LIN {X 0.053,Y -418.660,Z 515.534,A 0.000,B 0.000,C 90.000,E1 132.123} C_DIS
LIN {X -0.078,Y -417.973,Z 515.527,A 0.000,B 0.000,C 90.000,E1 130.782} C_DIS
LIN {X -0.019,Y -416.880,Z 515.517,A 0.000,B 0.000,C 90.000,E1 129.072} C_DIS
LIN {X -0.176,Y -415.818,Z 515.510,A 0.000,B 0.000,C 90.000,E1 127.729} C_DIS
LIN {X 0.148,Y -414.723,Z 515.501,A 0.000,B 0.000,C 90.000,E1 126.217} C_DIS
LIN {X 0.110,Y -414.727,Z 515.501,A 0.000,B 0.000,C 90.000,E1 126.217} C_DIS
LIN {X -0.098,Y -415.454,Z 515.500,A 0.000,B 0.000,C 90.000,E1 126.011} C_DIS
LIN {X -0.035,Y -425.850,Z 515.477,A 0.000,B 0.000,C 90.000,E1 121.926} C_DIS
LIN {X -0.091,Y -430.874,Z 515.468,A 0.000,B 0.000,C 90.000,E1 120.256} C_DIS
LIN {X -0.162,Y -439.919,Z 515.448,A 0.000,B 0.000,C 90.000,E1 116.616} C_DIS
LIN {X 0.024,Y -444.712,Z 515.439,A 0.000,B 0.000,C 90.000,E1 114.951} C_DIS
LIN {X -0.004,Y -454.683,Z 515.415,A 0.000,B 0.000,C 90.000,E1 110.737} C_DIS
LIN {X -0.228,Y -456.616,Z 515.411,A 0.000,B 0.000,C 90.000,E1 110.066} C_DIS
LIN {X -0.262,Y -456.708,Z 515.411,A 0.000,B 0.000,C 90.000,E1 110.066} C_DIS
LIN {X 0.078,Y -489.584,Z 515.405,A 0.000,B 0.000,C 90.000,E1 108.960} C_DIS
LIN {X 0.012,Y -503.421,Z 515.403,A 0.000,B 0.000,C 90.000,E1 108.489} C_DIS
LIN {X -0.146,Y -520.802,Z 515.399,A 0.000,B 0.000,C 90.000,E1 107.873} C_DIS
LIN {X -0.071,Y -534.501,Z 515.396,A 0.000,B 0.000,C 90.000,E1 107.330} C_DIS
LIN {X 0.020,Y -541.040,Z 515.395,A 0.000,B 0.000,C 90.000,E1 107.040} C_DIS
LIN {X 0.041,Y -547.560,Z 515.393,A 0.000,B 0.000,C 90.000,E1 106.732} C_DIS
LIN {X 0.199,Y -553.930,Z 515.391,A 0.000,B 0.000,C 90.000,E1 106.386} C_DIS
LIN {X -0.017,Y -559.838,Z 515.389,A 0.000,B 0.000,C 90.000,E1 106.079} C_DIS
LIN {X -0.116,Y -565.718,Z 515.387,A 0.000,B 0.000,C 90.000,E1 105.717} C_DIS
LIN {X -0.140,Y -571.713,Z 515.385,A 0.000,B 0.000,C 90.000,E1 105.300} C_DIS
LIN {X 0.274,Y -577.362,Z 515.383,A 0.000,B 0.000,C 90.000,E1 104.828} C_DIS
LIN {X -0.225,Y -582.899,Z 515.380,A 0.000,B 0.000,C 90.000,E1 104.411} C_DIS
LIN {X -0.192,Y -588.073,Z 515.377,A 0.000,B 0.000,C 90.000,E1 103.939} C_DIS
LIN {X 0.183,Y -593.940,Z 515.374,A 0.000,B 0.000,C 90.000,E1 103.300} C_DIS
LIN {X -0.050,Y -601.039,Z 515.370,A 0.000,B 0.000,C 90.000,E1 102.535} C_DIS
LIN {X 0.069,Y -605.510,Z 515.367,A 0.000,B 0.000,C 90.000,E1 102.007} C_DIS
LIN {X 0.219,Y -609.763,Z 515.364,A 0.000,B 0.000,C 90.000,E1 101.478} C_DIS
LIN {X 0.057,Y -615.614,Z 515.360,A 0.000,B 0.000,C 90.000,E1 100.715} C_DIS
LIN {X -0.165,Y -620.986,Z 515.355,A 0.000,B 0.000,C 90.000,E1 99.962} C_DIS
LIN {X 0.315,Y -624.961,Z 515.352,A 0.000,B 0.000,C 90.000,E1 99.321} C_DIS
LIN {X 0.189,Y -629.618,Z 515.348,A 0.000,B 0.000,C 90.000,E1 98.568} C_DIS
LIN {X 0.109,Y -633.925,Z 515.344,A 0.000,B 0.000,C 90.000,E1 97.814} C_DIS
LIN {X -0.201,Y -639.249,Z 515.338,A 0.000,B 0.000,C 90.000,E1 96.834} C_DIS
LIN {X -0.264,Y -642.915,Z 515.334,A 0.000,B 0.000,C 90.000,E1 96.087} C_DIS
LIN {X -0.054,Y -648.552,Z 515.327,A 0.000,B 0.000,C 90.000,E1 94.821} C_DIS
LIN {X -0.191,Y -652.488,Z 515.321,A 0.000,B 0.000,C 90.000,E1 93.841} C_DIS
LIN {X 0.041,Y -654.246,Z 515.319,A 0.000,B 0.000,C 90.000,E1 93.326} C_DIS
LIN {X 0.125,Y -656.498,Z 515.314,A 0.000,B 0.000,C 90.000,E1 92.579} C_DIS
LIN {X -0.263,Y -657.795,Z 515.312,A 0.000,B 0.000,C 90.000,E1 92.121} C_DIS
LIN {X 0.036,Y -658.865,Z 515.309,A 0.000,B 0.000,C 90.000,E1 91.604} C_DIS
LIN {X 0.139,Y -660.082,Z 515.305,A 0.000,B 0.000,C 90.000,E1 90.859} C_DIS
LIN {X -0.224,Y -660.593,Z 515.302,A 0.000,B 0.000,C 90.000,E1 90.401} C_DIS
LIN {X 0.256,Y -660.820,Z 515.301,A 0.000,B 0.000,C 90.000,E1 90.115} C_DIS
LIN {X -0.279,Y -660.960,Z 515.297,A 0.000,B 0.000,C 90.000,E1 89.427} C_DIS
LIN {X -0.154,Y -660.743,Z 515.293,A 0.000,B 0.000,C 90.000,E1 88.682} C_DIS
LIN {X -0.334,Y -660.657,Z 515.291,A 0.000,B 0.000,C 90.000,E1 88.453} C_DIS
LIN {X -0.193,Y -659.821,Z 515.287,A 0.000,B 0.000,C 90.000,E1 87.707} C_DIS
LIN {X 0.100,Y -659.109,Z 515.284,A 0.000,B 0.000,C 90.000,E1 87.192} C_DIS
LIN {X 0.231,Y -657.662,Z 515.280,A 0.000,B 0.000,C 90.000,E1 86.445} C_DIS
LIN {X 0.039,Y -657.169,Z 515.279,A 0.000,B 0.000,C 90.000,E1 86.216} C_DIS
LIN {X 0.152,Y -655.263,Z 515.275,A 0.000,B 0.000,C 90.000,E1 85.469} C_DIS
LIN {X -0.199,Y -653.811,Z 515.272,A 0.000,B 0.000,C 90.000,E1 85.008} C_DIS
LIN {X 0.095,Y -652.092,Z 515.269,A 0.000,B 0.000,C 90.000,E1 84.489} C_DIS
LIN {X -0.068,Y -648.360,Z 515.264,A 0.000,B 0.000,C 90.000,E1 83.514} C_DIS
LIN {X 0.026,Y -645.162,Z 515.260,A 0.000,B 0.000,C 90.000,E1 82.761} C_DIS
LIN {X 0.094,Y -641.550,Z 515.256,A 0.000,B 0.000,C 90.000,E1 82.008} C_DIS
LIN {X 0.124,Y -637.675,Z 515.252,A 0.000,B 0.000,C 90.000,E1 81.254} C_DIS
LIN {X 0.309,Y -634.940,Z 515.249,A 0.000,B 0.000,C 90.000,E1 80.735} C_DIS
LIN {X -0.208,Y -631.219,Z 515.245,A 0.000,B 0.000,C 90.000,E1 80.151} C_DIS
LIN {X -0.128,Y -627.261,Z 515.242,A 0.000,B 0.000,C 90.000,E1 79.511} C_DIS
LIN {X -0.083,Y -623.088,Z 515.238,A 0.000,B 0.000,C 90.000,E1 78.870} C_DIS
LIN {X -0.237,Y -616.739,Z 515.233,A 0.000,B 0.000,C 90.000,E1 77.993} C_DIS
LIN {X -0.288,Y -611.718,Z 515.230,A 0.000,B 0.000,C 90.000,E1 77.353} C_DIS
LIN {X -0.244,Y -606.038,Z 515.226,A 0.000,B 0.000,C 90.000,E1 76.700} C_DIS
LIN {X -0.133,Y -601.097,Z 515.223,A 0.000,B 0.000,C 90.000,E1 76.172} C_DIS
LIN {X 0.043,Y -595.900,Z 515.220,A 0.000,B 0.000,C 90.000,E1 75.644} C_DIS
LIN {X -0.173,Y -590.464,Z 515.218,A 0.000,B 0.000,C 90.000,E1 75.172} C_DIS
LIN {X -0.106,Y -584.679,Z 515.215,A 0.000,B 0.000,C 90.000,E1 74.685} C_DIS
LIN {X 0.133,Y -578.609,Z 515.212,A 0.000,B 0.000,C 90.000,E1 74.212} C_DIS
LIN {X 0.247,Y -572.611,Z 515.210,A 0.000,B 0.000,C 90.000,E1 73.795} C_DIS
LIN {X 0.100,Y -567.660,Z 515.208,A 0.000,B 0.000,C 90.000,E1 73.504} C_DIS
LIN {X -0.166,Y -562.686,Z 515.207,A 0.000,B 0.000,C 90.000,E1 73.251} C_DIS
LIN {X -0.083,Y -555.857,Z 515.205,A 0.000,B 0.000,C 90.000,E1 72.906} C_DIS
LIN {X 0.024,Y -548.840,Z 515.203,A 0.000,B 0.000,C 90.000,E1 72.598} C_DIS
LIN {X 0.259,Y -543.085,Z 515.202,A 0.000,B 0.000,C 90.000,E1 72.362} C_DIS
LIN {X -0.127,Y -538.051,Z 515.201,A 0.000,B 0.000,C 90.000,E1 72.236} C_DIS
LIN {X 0.029,Y -530.154,Z 515.200,A 0.000,B 0.000,C 90.000,E1 72.000} C_DIS
LIN {X -0.118,Y -524.165,Z 515.199,A 0.000,B 0.000,C 90.000,E1 71.873} C_DIS
LIN {X 0.066,Y -507.411,Z 515.197,A 0.000,B 0.000,C 90.000,E1 71.511} C_DIS
LIN {X -0.195,Y -499.131,Z 515.197,A 0.000,B 0.000,C 90.000,E1 71.402} C_DIS
LIN {X 0.111,Y -475.220,Z 515.195,A 0.000,B 0.000,C 90.000,E1 71.040} C_DIS
LIN {X -0.205,Y -472.091,Z 515.195,A 0.000,B 0.000,C 90.000,E1 71.040} C_DIS
LIN {X -0.231,Y -472.067,Z 515.195,A 0.000,B 0.000,C 90.000,E1 71.040} C_DIS
LIN {X 0.042,Y -465.715,Z 515.173,A 0.000,B 0.000,C 90.000,E1 67.102} C_DIS
LIN {X -0.162,Y -456.185,Z 515.146,A 0.000,B 0.000,C 90.000,E1 62.359} C_DIS
LIN {X -0.056,Y -455.669,Z 515.145,A 0.000,B 0.000,C 90.000,E1 62.025} C_DIS
LIN {X -0.064,Y -454.184,Z 515.141,A 0.000,B 0.000,C 90.000,E1 61.385} C_DIS
LIN {X 0.245,Y -447.007,Z 515.123,A 0.000,B 0.000,C 90.000,E1 58.122} C_DIS
LIN {X 0.205,Y -447.020,Z 515.123,A 0.000,B 0.000,C 90.000,E1 58.122} C_DIS
LIN {X 0.080,Y -449.700,Z 515.119,A 0.000,B 0.000,C 90.000,E1 57.375} C_DIS
LIN {X -0.057,Y -452.847,Z 515.113,A 0.000,B 0.000,C 90.000,E1 56.421} C_DIS
LIN {X -0.163,Y -455.733,Z 515.108,A 0.000,B 0.000,C 90.000,E1 55.468} C_DIS
LIN {X 0.022,Y -458.378,Z 515.103,A 0.000,B 0.000,C 90.000,E1 54.482} C_DIS
LIN {X -0.021,Y -461.358,Z 515.096,A 0.000,B 0.000,C 90.000,E1 53.210} C_DIS
LIN {X -0.139,Y -463.250,Z 515.090,A 0.000,B 0.000,C 90.000,E1 52.271} C_DIS
LIN {X 0.053,Y -464.835,Z 515.085,A 0.000,B 0.000,C 90.000,E1 51.295} C_DIS
LIN {X 0.030,Y -466.660,Z 515.078,A 0.000,B 0.000,C 90.000,E1 50.033} C_DIS
LIN {X -0.034,Y -467.855,Z 515.073,A 0.000,B 0.000,C 90.000,E1 49.094} C_DIS
LIN {X -0.063,Y -469.210,Z 515.066,A 0.000,B 0.000,C 90.000,E1 47.838} C_DIS
LIN {X -0.063,Y -470.270,Z 515.059,A 0.000,B 0.000,C 90.000,E1 46.581} C_DIS
LIN {X -0.136,Y -470.936,Z 515.054,A 0.000,B 0.000,C 90.000,E1 45.648} C_DIS
LIN {X 0.214,Y -471.520,Z 515.047,A 0.000,B 0.000,C 90.000,E1 44.352} C_DIS
LIN {X -0.277,Y -471.770,Z 515.043,A 0.000,B 0.000,C 90.000,E1 43.785} C_DIS
LIN {X -0.244,Y -471.920,Z 515.036,A 0.000,B 0.000,C 90.000,E1 42.528} C_DIS
LIN {X 0.140,Y -471.856,Z 515.029,A 0.000,B 0.000,C 90.000,E1 41.229} C_DIS
LIN {X 0.081,Y -471.672,Z 515.024,A 0.000,B 0.000,C 90.000,E1 40.297} C_DIS
LIN {X -0.072,Y -471.157,Z 515.015,A 0.000,B 0.000,C 90.000,E1 38.749} C_DIS
LIN {X 0.136,Y -470.405,Z 515.007,A 0.000,B 0.000,C 90.000,E1 37.156} C_DIS
LIN {X -0.178,Y -469.404,Z 514.996,A 0.000,B 0.000,C 90.000,E1 35.311} C_DIS
LIN {X -0.060,Y -468.652,Z 514.989,A 0.000,B 0.000,C 90.000,E1 34.040} C_DIS
LIN {X -0.067,Y -467.647,Z 514.980,A 0.000,B 0.000,C 90.000,E1 32.467} C_DIS
LIN {X -0.189,Y -466.304,Z 514.970,A 0.000,B 0.000,C 90.000,E1 30.590} C_DIS
LIN {X -0.089,Y -465.080,Z 514.961,A 0.000,B 0.000,C 90.000,E1 28.999} C_DIS
LIN {X 0.225,Y -463.394,Z 514.949,A 0.000,B 0.000,C 90.000,E1 26.744} C_DIS
LIN {X -0.246,Y -462.100,Z 514.938,A 0.000,B 0.000,C 90.000,E1 24.899} C_DIS
LIN {X 0.091,Y -460.907,Z 514.928,A 0.000,B 0.000,C 90.000,E1 22.950} C_DIS
LIN {X -0.037,Y -459.803,Z 514.915,A 0.000,B 0.000,C 90.000,E1 20.737} C_DIS
LIN {X -0.115,Y -459.061,Z 514.905,A 0.000,B 0.000,C 90.000,E1 18.833} C_DIS
LIN {X 0.035,Y -458.190,Z 514.890,A 0.000,B 0.000,C 90.000,E1 16.260} C_DIS
LIN {X 0.034,Y -457.764,Z 514.876,A 0.000,B 0.000,C 90.000,E1 13.703} C_DIS
LIN {X -0.080,Y -457.760,Z 514.864,A 0.000,B 0.000,C 90.000,E1 11.478} C_DIS
LIN {X -0.044,Y -458.183,Z 514.850,A 0.000,B 0.000,C 90.000,E1 8.916} C_DIS
LIN {X -0.185,Y -459.259,Z 514.832,A 0.000,B 0.000,C 90.000,E1 5.739} C_DIS
LIN {X 0.150,Y -460.241,Z 514.821,A 0.000,B 0.000,C 90.000,E1 3.784} C_DIS
LIN {X 0.215,Y -461.748,Z 514.809,A 0.000,B 0.000,C 90.000,E1 1.547} C_DIS
LIN {X 0.000,Y -463.039,Z 514.800,A 0.000,B 0.000,C 90.000,E1 360.000} C_DIS
LIN {X 0.072,Y -465.825,Z 514.785,A 0.000,B 0.000,C 90.000,E1 357.249} C_DIS
LIN {X 0.094,Y -468.899,Z 514.771,A 0.000,B 0.000,C 90.000,E1 354.723} C_DIS
LIN {X -0.031,Y -470.923,Z 514.762,A 0.000,B 0.000,C 90.000,E1 353.166} C_DIS
LIN {X -0.004,Y -473.942,Z 514.750,A 0.000,B 0.000,C 90.000,E1 350.971} C_DIS
LIN {X 0.098,Y -477.541,Z 514.736,A 0.000,B 0.000,C 90.000,E1 348.465} C_DIS
LIN {X 0.211,Y -483.309,Z 514.717,A 0.000,B 0.000,C 90.000,E1 345.046} C_DIS
LIN {X 0.132,Y -488.193,Z 514.703,A 0.000,B 0.000,C 90.000,E1 342.598} C_DIS
LIN {X -0.064,Y -491.366,Z 514.695,A 0.000,B 0.000,C 90.000,E1 341.094} C_DIS
LIN {X 0.000,Y -495.135,Z 514.685,A 0.000,B 0.000,C 90.000,E1 339.263} C_DIS
LIN {X 0.084,Y -498.253,Z 514.676,A 0.000,B 0.000,C 90.000,E1 337.741} C_DIS
LIN {X 0.211,Y -501.950,Z 514.666,A 0.000,B 0.000,C 90.000,E1 335.921} C_DIS
LIN {X -0.110,Y -504.840,Z 514.658,A 0.000,B 0.000,C 90.000,E1 334.460} C_DIS
LIN {X 0.070,Y -507.719,Z 514.650,A 0.000,B 0.000,C 90.000,E1 332.948} C_DIS
LIN {X -0.043,Y -511.253,Z 514.640,A 0.000,B 0.000,C 90.000,E1 331.179} C_DIS
LIN {X 0.196,Y -515.946,Z 514.627,A 0.000,B 0.000,C 90.000,E1 328.791} C_DIS
LIN {X 0.091,Y -519.587,Z 514.617,A 0.000,B 0.000,C 90.000,E1 327.041} C_DIS
LIN {X 0.251,Y -524.423,Z 514.604,A 0.000,B 0.000,C 90.000,E1 324.689} C_DIS
LIN {X 0.080,Y -527.432,Z 514.596,A 0.000,B 0.000,C 90.000,E1 323.256} C_DIS
LIN {X -0.037,Y -530.455,Z 514.588,A 0.000,B 0.000,C 90.000,E1 321.823} C_DIS
LIN {X -0.202,Y -534.629,Z 514.577,A 0.000,B 0.000,C 90.000,E1 319.828} C_DIS
LIN {X -0.280,Y -537.592,Z 514.569,A 0.000,B 0.000,C 90.000,E1 318.405} C_DIS
LIN {X 0.026,Y -541.239,Z 514.559,A 0.000,B 0.000,C 90.000,E1 316.662} C_DIS
LIN {X 0.029,Y -544.174,Z 514.551,A 0.000,B 0.000,C 90.000,E1 315.243} C_DIS
LIN {X -0.333,Y -545.817,Z 514.547,A 0.000,B 0.000,C 90.000,E1 314.433} C_DIS
LIN {X 0.158,Y -549.163,Z 514.537,A 0.000,B 0.000,C 90.000,E1 312.690} C_DIS
LIN {X 0.110,Y -554.500,Z 514.523,A 0.000,B 0.000,C 90.000,E1 310.172} C_DIS
LIN {X -0.306,Y -558.139,Z 514.514,A 0.000,B 0.000,C 90.000,E1 308.543} C_DIS
LIN {X 0.044,Y -560.372,Z 514.508,A 0.000,B 0.000,C 90.000,E1 307.397} C_DIS
LIN {X 0.181,Y -563.609,Z 514.499,A 0.000,B 0.000,C 90.000,E1 305.724} C_DIS
LIN {X 0.269,Y -570.539,Z 514.480,A 0.000,B 0.000,C 90.000,E1 302.418} C_DIS
LIN {X 0.116,Y -574.267,Z 514.471,A 0.000,B 0.000,C 90.000,E1 300.797} C_DIS
LIN {X -0.239,Y -576.738,Z 514.465,A 0.000,B 0.000,C 90.000,E1 299.745} C_DIS
LIN {X 0.304,Y -579.631,Z 514.460,A 0.000,B 0.000,C 90.000,E1 298.743} C_DIS
LIN {X 0.231,Y -580.359,Z 514.459,A 0.000,B 0.000,C 90.000,E1 298.615} C_DIS
LIN {X -0.157,Y -581.033,Z 514.458,A 0.000,B 0.000,C 90.000,E1 298.487} C_DIS
LIN {X -0.364,Y -582.119,Z 514.456,A 0.000,B 0.000,C 90.000,E1 298.103} C_DIS
LIN {X 0.355,Y -582.692,Z 514.455,A 0.000,B 0.000,C 90.000,E1 297.897} C_DIS
LIN {X 0.091,Y -583.563,Z 514.454,A 0.000,B 0.000,C 90.000,E1 297.769} C_DIS
LIN {X -0.039,Y -584.307,Z 514.453,A 0.000,B 0.000,C 90.000,E1 297.513} C_DIS
LIN {X -0.167,Y -584.833,Z 514.451,A 0.000,B 0.000,C 90.000,E1 297.257} C_DIS
LIN {X -0.292,Y -586.118,Z 514.450,A 0.000,B 0.000,C 90.000,E1 297.001} C_DIS
LIN {X 0.112,Y -586.668,Z 514.448,A 0.000,B 0.000,C 90.000,E1 296.693} C_DIS
LIN {X -0.120,Y -587.170,Z 514.445,A 0.000,B 0.000,C 90.000,E1 296.181} C_DIS
LIN {X -0.096,Y -587.929,Z 514.442,A 0.000,B 0.000,C 90.000,E1 295.643} C_DIS
LIN {X -0.056,Y -587.348,Z 514.438,A 0.000,B 0.000,C 90.000,E1 294.847} C_DIS
LIN {X -0.169,Y -586.947,Z 514.437,A 0.000,B 0.000,C 90.000,E1 294.591} C_DIS
LIN {X -0.284,Y -586.324,Z 514.435,A 0.000,B 0.000,C 90.000,E1 294.335} C_DIS
LIN {X 0.159,Y -584.433,Z 514.433,A 0.000,B 0.000,C 90.000,E1 293.898} C_DIS
LIN {X 0.116,Y -584.415,Z 514.433,A 0.000,B 0.000,C 90.000,E1 293.898} C_DIS
LIN {X -0.113,Y -583.588,Z 514.431,A 0.000,B 0.000,C 90.000,E1 293.515} C_DIS
LIN {X 0.277,Y -583.101,Z 514.428,A 0.000,B 0.000,C 90.000,E1 292.950} C_DIS
LIN {X 0.053,Y -583.102,Z 514.422,A 0.000,B 0.000,C 90.000,E1 291.897} C_DIS
LIN {X 0.289,Y -584.109,Z 514.411,A 0.000,B 0.000,C 90.000,E1 289.993} C_DIS
LIN {X 0.086,Y -584.451,Z 514.404,A 0.000,B 0.000,C 90.000,E1 288.671} C_DIS
LIN {X 0.230,Y -584.625,Z 514.398,A 0.000,B 0.000,C 90.000,E1 287.583} C_DIS
LIN {X 0.040,Y -584.599,Z 514.390,A 0.000,B 0.000,C 90.000,E1 286.260} C_DIS
LIN {X -0.024,Y -584.302,Z 514.378,A 0.000,B 0.000,C 90.000,E1 284.120} C_DIS
LIN {X -0.289,Y -584.056,Z 514.370,A 0.000,B 0.000,C 90.000,E1 282.535} C_DIS
LIN {X 0.013,Y -583.684,Z 514.361,A 0.000,B 0.000,C 90.000,E1 280.894} C_DIS
LIN {X -0.146,Y -583.228,Z 514.350,A 0.000,B 0.000,C 90.000,E1 279.029} C_DIS
LIN {X -0.074,Y -582.715,Z 514.341,A 0.000,B 0.000,C 90.000,E1 277.409} C_DIS
LIN {X -0.083,Y -582.139,Z 514.332,A 0.000,B 0.000,C 90.000,E1 275.796} C_DIS
LIN {X -0.154,Y -581.254,Z 514.323,A 0.000,B 0.000,C 90.000,E1 274.188} C_DIS
LIN {X 0.172,Y -580.310,Z 514.316,A 0.000,B 0.000,C 90.000,E1 272.808} C_DIS
LIN {X 0.276,Y -579.385,Z 514.310,A 0.000,B 0.000,C 90.000,E1 271.718} C_DIS
LIN {X -0.063,Y -578.193,Z 514.302,A 0.000,B 0.000,C 90.000,E1 270.401} C_DIS
LIN {X -0.263,Y -576.473,Z 514.293,A 0.000,B 0.000,C 90.000,E1 268.797} C_DIS
LIN {X 0.086,Y -574.673,Z 514.284,A 0.000,B 0.000,C 90.000,E1 267.135} C_DIS
LIN {X 0.289,Y -573.126,Z 514.277,A 0.000,B 0.000,C 90.000,E1 265.755} C_DIS
LIN {X 0.025,Y -571.189,Z 514.268,A 0.000,B 0.000,C 90.000,E1 264.147} C_DIS
LIN {X 0.226,Y -569.397,Z 514.260,A 0.000,B 0.000,C 90.000,E1 262.761} C_DIS
LIN {X -0.168,Y -567.404,Z 514.252,A 0.000,B 0.000,C 90.000,E1 261.432} C_DIS
LIN {X 0.216,Y -564.939,Z 514.243,A 0.000,B 0.000,C 90.000,E1 259.746} C_DIS
LIN {X 0.217,Y -563.319,Z 514.237,A 0.000,B 0.000,C 90.000,E1 258.645} C_DIS
LIN {X 0.030,Y -561.139,Z 514.229,A 0.000,B 0.000,C 90.000,E1 257.285} C_DIS
LIN {X 0.232,Y -558.850,Z 514.222,A 0.000,B 0.000,C 90.000,E1 255.880} C_DIS
LIN {X -0.024,Y -556.264,Z 514.214,A 0.000,B 0.000,C 90.000,E1 254.519} C_DIS
LIN {X 0.242,Y -554.069,Z 514.208,A 0.000,B 0.000,C 90.000,E1 253.378} C_DIS
LIN {X 0.058,Y -551.090,Z 514.200,A 0.000,B 0.000,C 90.000,E1 252.000} C_DIS
LIN {X -0.008,Y -547.915,Z 514.192,A 0.000,B 0.000,C 90.000,E1 250.604} C_DIS
LIN {X 0.065,Y -545.907,Z 514.188,A 0.000,B 0.000,C 90.000,E1 249.752} C_DIS
LIN {X 0.097,Y -542.424,Z 514.180,A 0.000,B 0.000,C 90.000,E1 248.337} C_DIS
LIN {X 0.062,Y -538.712,Z 514.172,A 0.000,B 0.000,C 90.000,E1 246.922} C_DIS
LIN {X -0.046,Y -535.590,Z 514.166,A 0.000,B 0.000,C 90.000,E1 245.793} C_DIS
LIN {X -0.007,Y -531.545,Z 514.158,A 0.000,B 0.000,C 90.000,E1 244.357} C_DIS
LIN {X 0.110,Y -526.503,Z 514.148,A 0.000,B 0.000,C 90.000,E1 242.615} C_DIS
LIN {X 0.048,Y -520.425,Z 514.137,A 0.000,B 0.000,C 90.000,E1 240.589} C_DIS
LIN {X -0.275,Y -515.161,Z 514.127,A 0.000,B 0.000,C 90.000,E1 238.869} C_DIS
LIN {X -0.084,Y -510.515,Z 514.119,A 0.000,B 0.000,C 90.000,E1 237.375} C_DIS
LIN {X 0.016,Y -505.735,Z 514.111,A 0.000,B 0.000,C 90.000,E1 235.881} C_DIS
LIN {X -0.190,Y -497.379,Z 514.096,A 0.000,B 0.000,C 90.000,E1 233.210} C_DIS
LIN {X -0.309,Y -490.497,Z 514.082,A 0.000,B 0.000,C 90.000,E1 230.803} C_DIS
LIN {X -0.013,Y -483.837,Z 514.068,A 0.000,B 0.000,C 90.000,E1 228.324} C_DIS
LIN {X 0.120,Y -478.990,Z 514.058,A 0.000,B 0.000,C 90.000,E1 226.458} C_DIS
LIN {X 0.023,Y -474.985,Z 514.050,A 0.000,B 0.000,C 90.000,E1 224.919} C_DIS
LIN {X -0.148,Y -471.100,Z 514.041,A 0.000,B 0.000,C 90.000,E1 223.380} C_DIS
LIN {X -0.127,Y -465.171,Z 514.027,A 0.000,B 0.000,C 90.000,E1 220.862} C_DIS
LIN {X 0.033,Y -460.167,Z 514.015,A 0.000,B 0.000,C 90.000,E1 218.624} C_DIS
LIN {X 0.023,Y -456.714,Z 514.006,A 0.000,B 0.000,C 90.000,E1 217.030} C_DIS
LIN {X -0.163,Y -451.350,Z 513.992,A 0.000,B 0.000,C 90.000,E1 214.485} C_DIS
LIN {X -0.099,Y -446.939,Z 513.979,A 0.000,B 0.000,C 90.000,E1 212.212} C_DIS
LIN {X -0.082,Y -443.264,Z 513.968,A 0.000,B 0.000,C 90.000,E1 210.256} C_DIS
LIN {X -0.169,Y -439.177,Z 513.955,A 0.000,B 0.000,C 90.000,E1 207.975} C_DIS
LIN {X -0.172,Y -435.119,Z 513.943,A 0.000,B 0.000,C 90.000,E1 205.668} C_DIS
LIN {X -0.082,Y -431.228,Z 513.930,A 0.000,B 0.000,C 90.000,E1 203.334} C_DIS
LIN {X 0.113,Y -427.465,Z 513.917,A 0.000,B 0.000,C 90.000,E1 200.972} C_DIS
LIN {X -0.094,Y -425.060,Z 513.907,A 0.000,B 0.000,C 90.000,E1 199.322} C_DIS
LIN {X 0.099,Y -422.293,Z 513.896,A 0.000,B 0.000,C 90.000,E1 197.275} C_DIS
LIN {X 0.103,Y -419.769,Z 513.885,A 0.000,B 0.000,C 90.000,E1 195.245} C_DIS
LIN {X -0.163,Y -417.298,Z 513.873,A 0.000,B 0.000,C 90.000,E1 193.244} C_DIS
LIN {X -0.030,Y -414.607,Z 513.860,A 0.000,B 0.000,C 90.000,E1 190.838} C_DIS
LIN {X 0.154,Y -413.162,Z 513.853,A 0.000,B 0.000,C 90.000,E1 189.443} C_DIS
LIN {X -0.027,Y -411.078,Z 513.841,A 0.000,B 0.000,C 90.000,E1 187.409} C_DIS
LIN {X 0.012,Y -408.521,Z 513.828,A 0.000,B 0.000,C 90.000,E1 184.992} C_DIS
LIN {X -0.179,Y -404.906,Z 513.803,A 0.000,B 0.000,C 90.000,E1 180.516} C_DIS
LIN {X -0.088,Y -402.866,Z 513.781,A 0.000,B 0.000,C 90.000,E1 176.674} C_DIS
LIN {X 0.038,Y -402.012,Z 513.762,A 0.000,B 0.000,C 90.000,E1 173.166} C_DIS
LIN {X -0.068,Y -401.958,Z 513.747,A 0.000,B 0.000,C 90.000,E1 170.387} C_DIS
LIN {X -0.041,Y -402.286,Z 513.731,A 0.000,B 0.000,C 90.000,E1 167.589} C_DIS
LIN {X -0.132,Y -403.037,Z 513.716,A 0.000,B 0.000,C 90.000,E1 164.810} C_DIS
LIN {X 0.117,Y -403.795,Z 513.706,A 0.000,B 0.000,C 90.000,E1 163.032} C_DIS
LIN {X -0.118,Y -405.419,Z 513.688,A 0.000,B 0.000,C 90.000,E1 159.934} C_DIS
LIN {X -0.093,Y -406.779,Z 513.677,A 0.000,B 0.000,C 90.000,E1 157.847} C_DIS
LIN {X 0.111,Y -407.794,Z 513.669,A 0.000,B 0.000,C 90.000,E1 156.433} C_DIS
LIN {X 0.034,Y -409.786,Z 513.656,A 0.000,B 0.000,C 90.000,E1 154.024} C_DIS
LIN {X -0.114,Y -410.870,Z 513.648,A 0.000,B 0.000,C 90.000,E1 152.666} C_DIS
LIN {X -0.022,Y -412.470,Z 513.637,A 0.000,B 0.000,C 90.000,E1 150.589} C_DIS
LIN {X 0.006,Y -413.632,Z 513.627,A 0.000,B 0.000,C 90.000,E1 148.869} C_DIS
LIN {X -0.080,Y -414.748,Z 513.618,A 0.000,B 0.000,C 90.000,E1 147.168} C_DIS
LIN {X -0.087,Y -415.629,Z 513.610,A 0.000,B 0.000,C 90.000,E1 145.801} C_DIS
LIN {X -0.062,Y -416.751,Z 513.599,A 0.000,B 0.000,C 90.000,E1 143.749} C_DIS
LIN {X 0.051,Y -417.617,Z 513.589,A 0.000,B 0.000,C 90.000,E1 142.029} C_DIS
LIN {X -0.155,Y -418.327,Z 513.580,A 0.000,B 0.000,C 90.000,E1 140.356} C_DIS
LIN {X -0.092,Y -418.961,Z 513.570,A 0.000,B 0.000,C 90.000,E1 138.647} C_DIS
LIN {X -0.252,Y -419.362,Z 513.563,A 0.000,B 0.000,C 90.000,E1 137.310} C_DIS
LIN {X 0.080,Y -419.617,Z 513.553,A 0.000,B 0.000,C 90.000,E1 135.567} C_DIS
LIN {X 0.227,Y -419.656,Z 513.546,A 0.000,B 0.000,C 90.000,E1 134.190} C_DIS
LIN {X 0.082,Y -419.468,Z 513.538,A 0.000,B 0.000,C 90.000,E1 132.852} C_DIS
LIN {X -0.147,Y -419.333,Z 513.534,A 0.000,B 0.000,C 90.000,E1 132.204} C_DIS
LIN {X 0.007,Y -418.624,Z 513.527,A 0.000,B 0.000,C 90.000,E1 130.825} C_DIS
LIN {X 0.069,Y -417.494,Z 513.517,A 0.000,B 0.000,C 90.000,E1 129.116} C_DIS
LIN {X -0.150,Y -416.150,Z 513.508,A 0.000,B 0.000,C 90.000,E1 127.443} C_DIS
LIN {X 0.141,Y -415.121,Z 513.501,A 0.000,B 0.000,C 90.000,E1 126.091} C_DIS
LIN {X 0.103,Y -415.120,Z 513.501,A 0.000,B 0.000,C 90.000,E1 126.091} C_DIS
LIN {X -0.131,Y -416.922,Z 513.497,A 0.000,B 0.000,C 90.000,E1 125.391} C_DIS
LIN {X -0.204,Y -426.654,Z 513.476,A 0.000,B 0.000,C 90.000,E1 121.671} C_DIS
LIN {X -0.242,Y -430.719,Z 513.468,A 0.000,B 0.000,C 90.000,E1 120.335} C_DIS
LIN {X 0.114,Y -440.681,Z 513.446,A 0.000,B 0.000,C 90.000,E1 116.309} C_DIS
LIN {X -0.123,Y -444.540,Z 513.439,A 0.000,B 0.000,C 90.000,E1 115.027} C_DIS
LIN {X 0.045,Y -446.679,Z 513.434,A 0.000,B 0.000,C 90.000,E1 114.027} C_DIS
LIN {X -0.089,Y -455.408,Z 513.414,A 0.000,B 0.000,C 90.000,E1 110.482} C_DIS
LIN {X -0.074,Y -457.381,Z 513.410,A 0.000,B 0.000,C 90.000,E1 109.758} C_DIS
LIN {X 0.031,Y -457.489,Z 513.409,A 0.000,B 0.000,C 90.000,E1 109.685} C_DIS
LIN {X -0.008,Y -457.632,Z 513.409,A 0.000,B 0.000,C 90.000,E1 109.685} C_DIS
LIN {X 0.093,Y -488.188,Z 513.404,A 0.000,B 0.000,C 90.000,E1 108.725} C_DIS
LIN {X -0.146,Y -501.969,Z 513.402,A 0.000,B 0.000,C 90.000,E1 108.290} C_DIS
LIN {X 0.177,Y -519.386,Z 513.398,A 0.000,B 0.000,C 90.000,E1 107.638} C_DIS
LIN {X 0.030,Y -526.157,Z 513.397,A 0.000,B 0.000,C 90.000,E1 107.402} C_DIS
LIN {X 0.154,Y -536.484,Z 513.395,A 0.000,B 0.000,C 90.000,E1 106.985} C_DIS
LIN {X -0.160,Y -542.966,Z 513.393,A 0.000,B 0.000,C 90.000,E1 106.732} C_DIS
LIN {X -0.135,Y -552.642,Z 513.390,A 0.000,B 0.000,C 90.000,E1 106.260} C_DIS
LIN {X 0.122,Y -558.921,Z 513.388,A 0.000,B 0.000,C 90.000,E1 105.898} C_DIS
LIN {X -0.059,Y -564.955,Z 513.386,A 0.000,B 0.000,C 90.000,E1 105.552} C_DIS
LIN {X 0.217,Y -570.715,Z 513.384,A 0.000,B 0.000,C 90.000,E1 105.134} C_DIS
LIN {X 0.201,Y -576.489,Z 513.382,A 0.000,B 0.000,C 90.000,E1 104.717} C_DIS
LIN {X 0.185,Y -582.988,Z 513.379,A 0.000,B 0.000,C 90.000,E1 104.189} C_DIS
LIN {X 0.198,Y -588.380,Z 513.376,A 0.000,B 0.000,C 90.000,E1 103.716} C_DIS
LIN {X -0.167,Y -594.543,Z 513.373,A 0.000,B 0.000,C 90.000,E1 103.119} C_DIS
LIN {X -0.139,Y -599.450,Z 513.370,A 0.000,B 0.000,C 90.000,E1 102.591} C_DIS
LIN {X -0.325,Y -605.228,Z 513.366,A 0.000,B 0.000,C 90.000,E1 101.951} C_DIS
LIN {X 0.026,Y -610.349,Z 513.363,A 0.000,B 0.000,C 90.000,E1 101.299} C_DIS
LIN {X -0.251,Y -616.399,Z 513.359,A 0.000,B 0.000,C 90.000,E1 100.546} C_DIS
LIN {X -0.292,Y -620.929,Z 513.355,A 0.000,B 0.000,C 90.000,E1 99.905} C_DIS
LIN {X -0.136,Y -624.526,Z 513.352,A 0.000,B 0.000,C 90.000,E1 99.378} C_DIS
LIN {X 0.014,Y -629.896,Z 513.347,A 0.000,B 0.000,C 90.000,E1 98.511} C_DIS
LIN {X 0.056,Y -634.261,Z 513.343,A 0.000,B 0.000,C 90.000,E1 97.757} C_DIS
LIN {X -0.249,Y -639.654,Z 513.338,A 0.000,B 0.000,C 90.000,E1 96.777} C_DIS
LIN {X -0.056,Y -642.169,Z 513.335,A 0.000,B 0.000,C 90.000,E1 96.258} C_DIS
LIN {X -0.267,Y -646.798,Z 513.329,A 0.000,B 0.000,C 90.000,E1 95.277} C_DIS
LIN {X -0.260,Y -650.093,Z 513.325,A 0.000,B 0.000,C 90.000,E1 94.531} C_DIS
LIN {X 0.224,Y -653.965,Z 513.320,A 0.000,B 0.000,C 90.000,E1 93.498} C_DIS
LIN {X 0.306,Y -656.310,Z 513.315,A 0.000,B 0.000,C 90.000,E1 92.751} C_DIS
LIN {X -0.276,Y -658.288,Z 513.311,A 0.000,B 0.000,C 90.000,E1 92.064} C_DIS
LIN {X 0.214,Y -658.890,Z 513.310,A 0.000,B 0.000,C 90.000,E1 91.776} C_DIS
LIN {X 0.316,Y -660.181,Z 513.306,A 0.000,B 0.000,C 90.000,E1 91.031} C_DIS
LIN {X -0.047,Y -660.825,Z 513.303,A 0.000,B 0.000,C 90.000,E1 90.573} C_DIS
LIN {X 0.257,Y -661.222,Z 513.300,A 0.000,B 0.000,C 90.000,E1 90.057} C_DIS
LIN {X -0.098,Y -661.329,Z 513.298,A 0.000,B 0.000,C 90.000,E1 89.599} C_DIS
LIN {X 0.031,Y -661.160,Z 513.294,A 0.000,B 0.000,C 90.000,E1 88.854} C_DIS
LIN {X -0.326,Y -660.900,Z 513.291,A 0.000,B 0.000,C 90.000,E1 88.396} C_DIS
LIN {X -0.002,Y -660.375,Z 513.288,A 0.000,B 0.000,C 90.000,E1 87.879} C_DIS
LIN {X 0.111,Y -659.215,Z 513.284,A 0.000,B 0.000,C 90.000,E1 87.135} C_DIS
LIN {X 0.243,Y -657.726,Z 513.280,A 0.000,B 0.000,C 90.000,E1 86.388} C_DIS
LIN {X 0.051,Y -657.205,Z 513.279,A 0.000,B 0.000,C 90.000,E1 86.159} C_DIS
LIN {X 0.164,Y -655.147,Z 513.275,A 0.000,B 0.000,C 90.000,E1 85.412} C_DIS
LIN {X -0.188,Y -653.622,Z 513.272,A 0.000,B 0.000,C 90.000,E1 84.951} C_DIS
LIN {X 0.105,Y -651.831,Z 513.269,A 0.000,B 0.000,C 90.000,E1 84.432} C_DIS
LIN {X 0.163,Y -648.894,Z 513.265,A 0.000,B 0.000,C 90.000,E1 83.685} C_DIS
LIN {X 0.264,Y -645.674,Z 513.261,A 0.000,B 0.000,C 90.000,E1 82.932} C_DIS
LIN {X -0.260,Y -642.715,Z 513.257,A 0.000,B 0.000,C 90.000,E1 82.356} C_DIS
LIN {X -0.219,Y -638.790,Z 513.253,A 0.000,B 0.000,C 90.000,E1 81.602} C_DIS
LIN {X -0.070,Y -634.005,Z 513.249,A 0.000,B 0.000,C 90.000,E1 80.735} C_DIS
LIN {X 0.223,Y -631.734,Z 513.246,A 0.000,B 0.000,C 90.000,E1 80.330} C_DIS
LIN {X 0.302,Y -627.751,Z 513.243,A 0.000,B 0.000,C 90.000,E1 79.690} C_DIS
LIN {X 0.140,Y -621.697,Z 513.238,A 0.000,B 0.000,C 90.000,E1 78.814} C_DIS
LIN {X 0.081,Y -616.097,Z 513.234,A 0.000,B 0.000,C 90.000,E1 78.049} C_DIS
LIN {X 0.027,Y -610.947,Z 513.230,A 0.000,B 0.000,C 90.000,E1 77.409} C_DIS
LIN {X 0.061,Y -605.053,Z 513.227,A 0.000,B 0.000,C 90.000,E1 76.756} C_DIS
LIN {X 0.217,Y -600.055,Z 513.224,A 0.000,B 0.000,C 90.000,E1 76.228} C_DIS
LIN {X -0.047,Y -593.586,Z 513.220,A 0.000,B 0.000,C 90.000,E1 75.644} C_DIS
LIN {X -0.027,Y -589.543,Z 513.218,A 0.000,B 0.000,C 90.000,E1 75.283} C_DIS
LIN {X 0.080,Y -583.818,Z 513.216,A 0.000,B 0.000,C 90.000,E1 74.810} C_DIS
LIN {X -0.127,Y -577.733,Z 513.213,A 0.000,B 0.000,C 90.000,E1 74.393} C_DIS
LIN {X -0.014,Y -571.566,Z 513.211,A 0.000,B 0.000,C 90.000,E1 73.976} C_DIS
LIN {X 0.015,Y -563.315,Z 513.208,A 0.000,B 0.000,C 90.000,E1 73.504} C_DIS
LIN {X 0.208,Y -556.427,Z 513.206,A 0.000,B 0.000,C 90.000,E1 73.142} C_DIS
LIN {X 0.096,Y -549.292,Z 513.205,A 0.000,B 0.000,C 90.000,E1 72.851} C_DIS
LIN {X -0.129,Y -543.625,Z 513.204,A 0.000,B 0.000,C 90.000,E1 72.670} C_DIS
LIN {X 0.080,Y -536.173,Z 513.202,A 0.000,B 0.000,C 90.000,E1 72.417} C_DIS
LIN {X -0.308,Y -530.590,Z 513.202,A 0.000,B 0.000,C 90.000,E1 72.308} C_DIS
LIN {X 0.081,Y -524.576,Z 513.201,A 0.000,B 0.000,C 90.000,E1 72.127} C_DIS
LIN {X 0.086,Y -507.521,Z 513.199,A 0.000,B 0.000,C 90.000,E1 71.819} C_DIS
LIN {X 0.275,Y -497.747,Z 513.198,A 0.000,B 0.000,C 90.000,E1 71.638} C_DIS
LIN {X -0.032,Y -485.055,Z 513.197,A 0.000,B 0.000,C 90.000,E1 71.511} C_DIS
LIN {X -0.257,Y -472.933,Z 513.197,A 0.000,B 0.000,C 90.000,E1 71.402} C_DIS
LIN {X -0.282,Y -472.767,Z 513.197,A 0.000,B 0.000,C 90.000,E1 71.402} C_DIS
LIN {X 0.226,Y -465.916,Z 513.174,A 0.000,B 0.000,C 90.000,E1 67.230} C_DIS
LIN {X 0.168,Y -465.392,Z 513.172,A 0.000,B 0.000,C 90.000,E1 66.922} C_DIS
LIN {X -0.073,Y -456.977,Z 513.149,A 0.000,B 0.000,C 90.000,E1 62.820} C_DIS
LIN {X 0.032,Y -455.375,Z 513.144,A 0.000,B 0.000,C 90.000,E1 61.847} C_DIS
LIN {X 0.001,Y -447.354,Z 513.124,A 0.000,B 0.000,C 90.000,E1 58.329} C_DIS
LIN {X -0.040,Y -447.371,Z 513.124,A 0.000,B 0.000,C 90.000,E1 58.329} C_DIS
LIN {X -0.053,Y -449.868,Z 513.120,A 0.000,B 0.000,C 90.000,E1 57.661} C_DIS
LIN {X -0.190,Y -453.154,Z 513.115,A 0.000,B 0.000,C 90.000,E1 56.707} C_DIS
LIN {X -0.037,Y -456.173,Z 513.110,A 0.000,B 0.000,C 90.000,E1 55.722} C_DIS
LIN {X -0.106,Y -458.943,Z 513.104,A 0.000,B 0.000,C 90.000,E1 54.769} C_DIS
LIN {X -0.142,Y -462.004,Z 513.097,A 0.000,B 0.000,C 90.000,E1 53.497} C_DIS
LIN {X -0.003,Y -463.344,Z 513.094,A 0.000,B 0.000,C 90.000,E1 52.844} C_DIS
LIN {X 0.149,Y -464.545,Z 513.090,A 0.000,B 0.000,C 90.000,E1 52.190} C_DIS
LIN {X 0.067,Y -466.081,Z 513.085,A 0.000,B 0.000,C 90.000,E1 51.251} C_DIS
LIN {X 0.058,Y -467.859,Z 513.078,A 0.000,B 0.000,C 90.000,E1 49.989} C_DIS
LIN {X -0.045,Y -469.032,Z 513.073,A 0.000,B 0.000,C 90.000,E1 49.057} C_DIS
LIN {X -0.015,Y -470.321,Z 513.066,A 0.000,B 0.000,C 90.000,E1 47.796} C_DIS
LIN {X -0.007,Y -471.316,Z 513.059,A 0.000,B 0.000,C 90.000,E1 46.539} C_DIS
LIN {X 0.258,Y -471.930,Z 513.053,A 0.000,B 0.000,C 90.000,E1 45.567} C_DIS
LIN {X -0.136,Y -472.381,Z 513.048,A 0.000,B 0.000,C 90.000,E1 44.676} C_DIS
LIN {X 0.141,Y -472.704,Z 513.043,A 0.000,B 0.000,C 90.000,E1 43.704} C_DIS
LIN {X 0.187,Y -472.820,Z 513.036,A 0.000,B 0.000,C 90.000,E1 42.447} C_DIS
LIN {X -0.082,Y -472.712,Z 513.029,A 0.000,B 0.000,C 90.000,E1 41.229} C_DIS
LIN {X 0.009,Y -472.405,Z 513.022,A 0.000,B 0.000,C 90.000,E1 39.967} C_DIS
LIN {X 0.173,Y -471.792,Z 513.013,A 0.000,B 0.000,C 90.000,E1 38.382} C_DIS
LIN {X -0.266,Y -471.000,Z 513.005,A 0.000,B 0.000,C 90.000,E1 36.870} C_DIS
LIN {X 0.087,Y -469.971,Z 512.994,A 0.000,B 0.000,C 90.000,E1 34.945} C_DIS
LIN {X -0.127,Y -468.751,Z 512.984,A 0.000,B 0.000,C 90.000,E1 33.086} C_DIS
LIN {X 0.265,Y -467.619,Z 512.975,A 0.000,B 0.000,C 90.000,E1 31.465} C_DIS
LIN {X -0.009,Y -466.437,Z 512.966,A 0.000,B 0.000,C 90.000,E1 29.922} C_DIS
LIN {X 0.009,Y -464.904,Z 512.956,A 0.000,B 0.000,C 90.000,E1 28.025} C_DIS
LIN {X 0.188,Y -463.493,Z 512.945,A 0.000,B 0.000,C 90.000,E1 26.104} C_DIS
LIN {X 0.212,Y -462.399,Z 512.936,A 0.000,B 0.000,C 90.000,E1 24.515} C_DIS
LIN {X -0.055,Y -461.214,Z 512.926,A 0.000,B 0.000,C 90.000,E1 22.642} C_DIS
LIN {X -0.094,Y -460.270,Z 512.915,A 0.000,B 0.000,C 90.000,E1 20.737} C_DIS
LIN {X 0.275,Y -459.499,Z 512.905,A 0.000,B 0.000,C 90.000,E1 18.779} C_DIS
LIN {X 0.002,Y -458.570,Z 512.890,A 0.000,B 0.000,C 90.000,E1 16.260} C_DIS
LIN {X 0.013,Y -458.100,Z 512.876,A 0.000,B 0.000,C 90.000,E1 13.703} C_DIS
LIN {X -0.092,Y -458.080,Z 512.864,A 0.000,B 0.000,C 90.000,E1 11.478} C_DIS
LIN {X -0.047,Y -458.459,Z 512.850,A 0.000,B 0.000,C 90.000,E1 8.916} C_DIS
LIN {X -0.177,Y -459.497,Z 512.832,A 0.000,B 0.000,C 90.000,E1 5.739} C_DIS
LIN {X 0.163,Y -460.457,Z 512.821,A 0.000,B 0.000,C 90.000,E1 3.784} C_DIS
LIN {X 0.234,Y -461.940,Z 512.809,A 0.000,B 0.000,C 90.000,E1 1.547} C_DIS
LIN {X 0.000,Y -463.227,Z 512.800,A 0.000,B 0.000,C 90.000,E1 360.000} C_DIS
LIN {X 0.078,Y -465.986,Z 512.785,A 0.000,B 0.000,C 90.000,E1 357.249} C_DIS
LIN {X -0.093,Y -469.470,Z 512.769,A 0.000,B 0.000,C 90.000,E1 354.432} C_DIS
LIN {X -0.157,Y -472.315,Z 512.757,A 0.000,B 0.000,C 90.000,E1 352.243} C_DIS
LIN {X -0.156,Y -474.479,Z 512.748,A 0.000,B 0.000,C 90.000,E1 350.679} C_DIS
LIN {X -0.037,Y -478.128,Z 512.734,A 0.000,B 0.000,C 90.000,E1 348.173} C_DIS
LIN {X 0.087,Y -484.649,Z 512.714,A 0.000,B 0.000,C 90.000,E1 344.448} C_DIS
LIN {X 0.163,Y -488.369,Z 512.703,A 0.000,B 0.000,C 90.000,E1 342.598} C_DIS
LIN {X 0.002,Y -492.190,Z 512.693,A 0.000,B 0.000,C 90.000,E1 340.786} C_DIS
LIN {X 0.089,Y -495.992,Z 512.683,A 0.000,B 0.000,C 90.000,E1 338.954} C_DIS
LIN {X -0.275,Y -499.114,Z 512.675,A 0.000,B 0.000,C 90.000,E1 337.486} C_DIS
LIN {X -0.125,Y -502.792,Z 512.665,A 0.000,B 0.000,C 90.000,E1 335.665} C_DIS
LIN {X 0.024,Y -505.675,Z 512.656,A 0.000,B 0.000,C 90.000,E1 334.152} C_DIS
LIN {X 0.129,Y -508.015,Z 512.650,A 0.000,B 0.000,C 90.000,E1 332.948} C_DIS
LIN {X 0.114,Y -512.139,Z 512.638,A 0.000,B 0.000,C 90.000,E1 330.873} C_DIS
LIN {X 0.006,Y -516.318,Z 512.627,A 0.000,B 0.000,C 90.000,E1 328.820} C_DIS
LIN {X 0.117,Y -520.574,Z 512.615,A 0.000,B 0.000,C 90.000,E1 326.755} C_DIS
LIN {X -0.079,Y -524.868,Z 512.604,A 0.000,B 0.000,C 90.000,E1 324.736} C_DIS
LIN {X -0.129,Y -527.945,Z 512.596,A 0.000,B 0.000,C 90.000,E1 323.290} C_DIS
LIN {X 0.065,Y -531.566,Z 512.586,A 0.000,B 0.000,C 90.000,E1 321.537} C_DIS
LIN {X -0.070,Y -535.193,Z 512.577,A 0.000,B 0.000,C 90.000,E1 319.828} C_DIS
LIN {X -0.137,Y -538.202,Z 512.569,A 0.000,B 0.000,C 90.000,E1 318.405} C_DIS
LIN {X -0.189,Y -541.859,Z 512.559,A 0.000,B 0.000,C 90.000,E1 316.701} C_DIS
LIN {X -0.179,Y -545.368,Z 512.550,A 0.000,B 0.000,C 90.000,E1 315.000} C_DIS
LIN {X -0.093,Y -548.753,Z 512.541,A 0.000,B 0.000,C 90.000,E1 313.299} C_DIS
LIN {X -0.224,Y -553.337,Z 512.528,A 0.000,B 0.000,C 90.000,E1 311.067} C_DIS
LIN {X 0.041,Y -556.297,Z 512.520,A 0.000,B 0.000,C 90.000,E1 309.644} C_DIS
LIN {X -0.077,Y -558.749,Z 512.514,A 0.000,B 0.000,C 90.000,E1 308.543} C_DIS
LIN {X -0.161,Y -561.031,Z 512.508,A 0.000,B 0.000,C 90.000,E1 307.443} C_DIS
LIN {X -0.244,Y -564.818,Z 512.497,A 0.000,B 0.000,C 90.000,E1 305.518} C_DIS
LIN {X 0.023,Y -569.340,Z 512.485,A 0.000,B 0.000,C 90.000,E1 303.293} C_DIS
LIN {X 0.018,Y -572.341,Z 512.477,A 0.000,B 0.000,C 90.000,E1 301.926} C_DIS
LIN {X -0.241,Y -575.164,Z 512.470,A 0.000,B 0.000,C 90.000,E1 300.590} C_DIS
LIN {X 0.048,Y -578.031,Z 512.462,A 0.000,B 0.000,C 90.000,E1 299.205} C_DIS
LIN {X -0.247,Y -579.209,Z 512.459,A 0.000,B 0.000,C 90.000,E1 298.693} C_DIS
LIN {X -0.067,Y -580.098,Z 512.458,A 0.000,B 0.000,C 90.000,E1 298.409} C_DIS
LIN {X -0.106,Y -582.946,Z 512.452,A 0.000,B 0.000,C 90.000,E1 297.334} C_DIS
LIN {X -0.100,Y -584.218,Z 512.449,A 0.000,B 0.000,C 90.000,E1 296.796} C_DIS
LIN {X -0.193,Y -585.588,Z 512.444,A 0.000,B 0.000,C 90.000,E1 295.848} C_DIS
LIN {X -0.026,Y -585.898,Z 512.439,A 0.000,B 0.000,C 90.000,E1 295.027} C_DIS
LIN {X -0.146,Y -585.702,Z 512.438,A 0.000,B 0.000,C 90.000,E1 294.771} C_DIS
LIN {X -0.267,Y -585.334,Z 512.436,A 0.000,B 0.000,C 90.000,E1 294.515} C_DIS
LIN {X 0.145,Y -584.674,Z 512.435,A 0.000,B 0.000,C 90.000,E1 294.207} C_DIS
LIN {X 0.022,Y -584.669,Z 512.433,A 0.000,B 0.000,C 90.000,E1 293.951} C_DIS
LIN {X 0.303,Y -584.238,Z 512.430,A 0.000,B 0.000,C 90.000,E1 293.387} C_DIS
LIN {X -0.112,Y -584.042,Z 512.427,A 0.000,B 0.000,C 90.000,E1 292.898} C_DIS
LIN {X -0.318,Y -584.230,Z 512.421,A 0.000,B 0.000,C 90.000,E1 291.844} C_DIS
LIN {X 0.091,Y -585.200,Z 512.412,A 0.000,B 0.000,C 90.000,E1 290.194} C_DIS
LIN {X 0.106,Y -585.628,Z 512.405,A 0.000,B 0.000,C 90.000,E1 288.852} C_DIS
LIN {X -0.290,Y -585.827,Z 512.399,A 0.000,B 0.000,C 90.000,E1 287.819} C_DIS
LIN {X 0.100,Y -585.852,Z 512.391,A 0.000,B 0.000,C 90.000,E1 286.441} C_DIS
LIN {X 0.076,Y -585.675,Z 512.380,A 0.000,B 0.000,C 90.000,E1 284.300} C_DIS
LIN {X 0.217,Y -585.399,Z 512.369,A 0.000,B 0.000,C 90.000,E1 282.411} C_DIS
LIN {X 0.182,Y -585.144,Z 512.362,A 0.000,B 0.000,C 90.000,E1 281.074} C_DIS
LIN {X 0.067,Y -584.723,Z 512.351,A 0.000,B 0.000,C 90.000,E1 279.208} C_DIS
LIN {X 0.022,Y -584.357,Z 512.344,A 0.000,B 0.000,C 90.000,E1 277.871} C_DIS
LIN {X -0.118,Y -583.864,Z 512.336,A 0.000,B 0.000,C 90.000,E1 276.543} C_DIS
LIN {X 0.029,Y -583.433,Z 512.330,A 0.000,B 0.000,C 90.000,E1 275.454} C_DIS
LIN {X -0.179,Y -582.659,Z 512.323,A 0.000,B 0.000,C 90.000,E1 274.131} C_DIS
LIN {X 0.172,Y -581.705,Z 512.315,A 0.000,B 0.000,C 90.000,E1 272.751} C_DIS
LIN {X 0.108,Y -581.005,Z 512.311,A 0.000,B 0.000,C 90.000,E1 271.949} C_DIS
LIN {X -0.187,Y -579.768,Z 512.303,A 0.000,B 0.000,C 90.000,E1 270.630} C_DIS
LIN {X 0.225,Y -578.050,Z 512.294,A 0.000,B 0.000,C 90.000,E1 268.969} C_DIS
LIN {X 0.182,Y -575.894,Z 512.284,A 0.000,B 0.000,C 90.000,E1 267.078} C_DIS
LIN {X 0.225,Y -574.638,Z 512.278,A 0.000,B 0.000,C 90.000,E1 265.988} C_DIS
LIN {X 0.038,Y -572.644,Z 512.269,A 0.000,B 0.000,C 90.000,E1 264.375} C_DIS
LIN {X 0.200,Y -570.829,Z 512.261,A 0.000,B 0.000,C 90.000,E1 262.996} C_DIS
LIN {X -0.094,Y -568.799,Z 512.254,A 0.000,B 0.000,C 90.000,E1 261.659} C_DIS
LIN {X -0.152,Y -565.860,Z 512.243,A 0.000,B 0.000,C 90.000,E1 259.746} C_DIS
LIN {X 0.141,Y -563.733,Z 512.235,A 0.000,B 0.000,C 90.000,E1 258.342} C_DIS
LIN {X -0.151,Y -561.463,Z 512.228,A 0.000,B 0.000,C 90.000,E1 256.992} C_DIS
LIN {X -0.091,Y -559.607,Z 512.222,A 0.000,B 0.000,C 90.000,E1 255.880} C_DIS
LIN {X -0.332,Y -556.971,Z 512.214,A 0.000,B 0.000,C 90.000,E1 254.519} C_DIS
LIN {X -0.055,Y -554.733,Z 512.208,A 0.000,B 0.000,C 90.000,E1 253.378} C_DIS
LIN {X -0.225,Y -551.714,Z 512.200,A 0.000,B 0.000,C 90.000,E1 252.000} C_DIS
LIN {X 0.239,Y -548.509,Z 512.192,A 0.000,B 0.000,C 90.000,E1 250.550} C_DIS
LIN {X 0.059,Y -545.765,Z 512.186,A 0.000,B 0.000,C 90.000,E1 249.444} C_DIS
LIN {X -0.155,Y -542.924,Z 512.180,A 0.000,B 0.000,C 90.000,E1 248.337} C_DIS
LIN {X -0.179,Y -539.197,Z 512.172,A 0.000,B 0.000,C 90.000,E1 246.922} C_DIS
LIN {X -0.067,Y -535.245,Z 512.164,A 0.000,B 0.000,C 90.000,E1 245.485} C_DIS
LIN {X 0.191,Y -531.106,Z 512.156,A 0.000,B 0.000,C 90.000,E1 244.024} C_DIS
LIN {X -0.102,Y -526.860,Z 512.148,A 0.000,B 0.000,C 90.000,E1 242.615} C_DIS
LIN {X 0.168,Y -521.627,Z 512.138,A 0.000,B 0.000,C 90.000,E1 240.845} C_DIS
LIN {X -0.127,Y -516.360,Z 512.128,A 0.000,B 0.000,C 90.000,E1 239.125} C_DIS
LIN {X -0.185,Y -511.724,Z 512.120,A 0.000,B 0.000,C 90.000,E1 237.661} C_DIS
LIN {X 0.314,Y -507.951,Z 512.114,A 0.000,B 0.000,C 90.000,E1 236.421} C_DIS
LIN {X 0.127,Y -501.251,Z 512.102,A 0.000,B 0.000,C 90.000,E1 234.356} C_DIS
LIN {X -0.055,Y -494.921,Z 512.090,A 0.000,B 0.000,C 90.000,E1 232.271} C_DIS
LIN {X 0.068,Y -489.796,Z 512.080,A 0.000,B 0.000,C 90.000,E1 230.436} C_DIS
LIN {X -0.165,Y -483.972,Z 512.068,A 0.000,B 0.000,C 90.000,E1 228.324} C_DIS
LIN {X -0.151,Y -479.967,Z 512.060,A 0.000,B 0.000,C 90.000,E1 226.782} C_DIS
LIN {X -0.119,Y -475.106,Z 512.049,A 0.000,B 0.000,C 90.000,E1 224.919} C_DIS
LIN {X 0.055,Y -471.202,Z 512.041,A 0.000,B 0.000,C 90.000,E1 223.338} C_DIS
LIN {X -0.020,Y -466.006,Z 512.029,A 0.000,B 0.000,C 90.000,E1 221.148} C_DIS
LIN {X -0.098,Y -460.272,Z 512.015,A 0.000,B 0.000,C 90.000,E1 218.624} C_DIS
LIN {X -0.104,Y -456.824,Z 512.006,A 0.000,B 0.000,C 90.000,E1 217.030} C_DIS
LIN {X -0.030,Y -451.486,Z 511.991,A 0.000,B 0.000,C 90.000,E1 214.452} C_DIS
LIN {X -0.216,Y -447.078,Z 511.979,A 0.000,B 0.000,C 90.000,E1 212.212} C_DIS
LIN {X 0.187,Y -443.425,Z 511.968,A 0.000,B 0.000,C 90.000,E1 210.207} C_DIS
LIN {X -0.276,Y -439.337,Z 511.955,A 0.000,B 0.000,C 90.000,E1 207.975} C_DIS
LIN {X -0.103,Y -435.843,Z 511.944,A 0.000,B 0.000,C 90.000,E1 205.976} C_DIS
LIN {X 0.002,Y -431.931,Z 511.931,A 0.000,B 0.000,C 90.000,E1 203.643} C_DIS
LIN {X 0.215,Y -428.083,Z 511.918,A 0.000,B 0.000,C 90.000,E1 201.280} C_DIS
LIN {X 0.216,Y -425.129,Z 511.907,A 0.000,B 0.000,C 90.000,E1 199.268} C_DIS
LIN {X -0.172,Y -422.814,Z 511.898,A 0.000,B 0.000,C 90.000,E1 197.638} C_DIS
LIN {X 0.017,Y -419.818,Z 511.885,A 0.000,B 0.000,C 90.000,E1 195.245} C_DIS
LIN {X -0.152,Y -417.351,Z 511.873,A 0.000,B 0.000,C 90.000,E1 193.231} C_DIS
LIN {X -0.161,Y -415.033,Z 511.862,A 0.000,B 0.000,C 90.000,E1 191.186} C_DIS
LIN {X 0.073,Y -413.214,Z 511.853,A 0.000,B 0.000,C 90.000,E1 189.443} C_DIS
LIN {X -0.106,Y -411.131,Z 511.841,A 0.000,B 0.000,C 90.000,E1 187.409} C_DIS
LIN {X -0.046,Y -408.957,Z 511.830,A 0.000,B 0.000,C 90.000,E1 185.334} C_DIS
LIN {X 0.153,Y -404.980,Z 511.803,A 0.000,B 0.000,C 90.000,E1 180.458} C_DIS
LIN {X -0.156,Y -402.943,Z 511.781,A 0.000,B 0.000,C 90.000,E1 176.674} C_DIS
LIN {X -0.020,Y -402.146,Z 511.764,A 0.000,B 0.000,C 90.000,E1 173.514} C_DIS
LIN {X -0.130,Y -402.052,Z 511.747,A 0.000,B 0.000,C 90.000,E1 170.387} C_DIS
LIN {X -0.101,Y -402.410,Z 511.731,A 0.000,B 0.000,C 90.000,E1 167.589} C_DIS
LIN {X -0.187,Y -403.174,Z 511.716,A 0.000,B 0.000,C 90.000,E1 164.810} C_DIS
LIN {X -0.224,Y -404.073,Z 511.704,A 0.000,B 0.000,C 90.000,E1 162.725} C_DIS
LIN {X -0.165,Y -405.600,Z 511.688,A 0.000,B 0.000,C 90.000,E1 159.934} C_DIS
LIN {X -0.030,Y -407.221,Z 511.675,A 0.000,B 0.000,C 90.000,E1 157.486} C_DIS
LIN {X -0.026,Y -408.813,Z 511.663,A 0.000,B 0.000,C 90.000,E1 155.409} C_DIS
LIN {X 0.000,Y -410.027,Z 511.656,A 0.000,B 0.000,C 90.000,E1 154.024} C_DIS
LIN {X -0.144,Y -411.115,Z 511.648,A 0.000,B 0.000,C 90.000,E1 152.666} C_DIS
LIN {X 0.022,Y -412.478,Z 511.639,A 0.000,B 0.000,C 90.000,E1 150.923} C_DIS
LIN {X 0.051,Y -413.741,Z 511.629,A 0.000,B 0.000,C 90.000,E1 149.203} C_DIS
LIN {X -0.033,Y -414.906,Z 511.619,A 0.000,B 0.000,C 90.000,E1 147.502} C_DIS
LIN {X -0.092,Y -416.006,Z 511.610,A 0.000,B 0.000,C 90.000,E1 145.801} C_DIS
LIN {X -0.116,Y -417.394,Z 511.597,A 0.000,B 0.000,C 90.000,E1 143.417} C_DIS
LIN {X 0.000,Y -418.279,Z 511.587,A 0.000,B 0.000,C 90.000,E1 141.698} C_DIS
LIN {X 0.065,Y -419.034,Z 511.578,A 0.000,B 0.000,C 90.000,E1 139.989} C_DIS
LIN {X -0.175,Y -419.668,Z 511.568,A 0.000,B 0.000,C 90.000,E1 138.324} C_DIS
LIN {X -0.013,Y -420.069,Z 511.561,A 0.000,B 0.000,C 90.000,E1 136.944} C_DIS
LIN {X 0.028,Y -420.290,Z 511.551,A 0.000,B 0.000,C 90.000,E1 135.243} C_DIS
LIN {X 0.185,Y -420.311,Z 511.544,A 0.000,B 0.000,C 90.000,E1 133.866} C_DIS
LIN {X 0.049,Y -420.074,Z 511.536,A 0.000,B 0.000,C 90.000,E1 132.528} C_DIS
LIN {X 0.020,Y -419.696,Z 511.531,A 0.000,B 0.000,C 90.000,E1 131.515} C_DIS
LIN {X -0.092,Y -418.840,Z 511.523,A 0.000,B 0.000,C 90.000,E1 130.172} C_DIS
LIN {X 0.177,Y -418.088,Z 511.517,A 0.000,B 0.000,C 90.000,E1 129.116} C_DIS
LIN {X -0.031,Y -416.749,Z 511.508,A 0.000,B 0.000,C 90.000,E1 127.443} C_DIS
LIN {X 0.026,Y -415.552,Z 511.500,A 0.000,B 0.000,C 90.000,E1 125.964} C_DIS
LIN {X -0.012,Y -415.557,Z 511.500,A 0.000,B 0.000,C 90.000,E1 125.964} C_DIS
LIN {X -0.050,Y -425.629,Z 511.478,A 0.000,B 0.000,C 90.000,E1 122.005} C_DIS
LIN {X -0.106,Y -430.666,Z 511.469,A 0.000,B 0.000,C 90.000,E1 120.335} C_DIS
LIN {X -0.145,Y -440.631,Z 511.446,A 0.000,B 0.000,C 90.000,E1 116.360} C_DIS
LIN {X 0.014,Y -444.486,Z 511.439,A 0.000,B 0.000,C 90.000,E1 115.027} C_DIS
LIN {X -0.088,Y -445.947,Z 511.435,A 0.000,B 0.000,C 90.000,E1 114.387} C_DIS
LIN {X 0.049,Y -455.360,Z 511.414,A 0.000,B 0.000,C 90.000,E1 110.482} C_DIS
LIN {X 0.273,Y -457.159,Z 511.410,A 0.000,B 0.000,C 90.000,E1 109.812} C_DIS
LIN {X 0.224,Y -458.094,Z 511.408,A 0.000,B 0.000,C 90.000,E1 109.322} C_DIS
LIN {X 0.184,Y -458.170,Z 511.408,A 0.000,B 0.000,C 90.000,E1 109.322} C_DIS
LIN {X -0.148,Y -487.720,Z 511.403,A 0.000,B 0.000,C 90.000,E1 108.471} C_DIS
LIN {X 0.056,Y -501.510,Z 511.400,A 0.000,B 0.000,C 90.000,E1 108.000} C_DIS
LIN {X 0.169,Y -515.430,Z 511.397,A 0.000,B 0.000,C 90.000,E1 107.511} C_DIS
LIN {X 0.086,Y -522.414,Z 511.396,A 0.000,B 0.000,C 90.000,E1 107.275} C_DIS
LIN {X 0.163,Y -536.058,Z 511.393,A 0.000,B 0.000,C 90.000,E1 106.749} C_DIS
LIN {X -0.054,Y -542.587,Z 511.392,A 0.000,B 0.000,C 90.000,E1 106.496} C_DIS
LIN {X 0.107,Y -552.391,Z 511.389,A 0.000,B 0.000,C 90.000,E1 106.024} C_DIS
LIN {X -0.128,Y -558.678,Z 511.387,A 0.000,B 0.000,C 90.000,E1 105.717} C_DIS
LIN {X -0.146,Y -564.605,Z 511.385,A 0.000,B 0.000,C 90.000,E1 105.371} C_DIS
LIN {X 0.121,Y -570.517,Z 511.383,A 0.000,B 0.000,C 90.000,E1 104.954} C_DIS
LIN {X 0.111,Y -576.374,Z 511.381,A 0.000,B 0.000,C 90.000,E1 104.537} C_DIS
LIN {X -0.124,Y -581.951,Z 511.378,A 0.000,B 0.000,C 90.000,E1 104.120} C_DIS
LIN {X 0.018,Y -587.337,Z 511.376,A 0.000,B 0.000,C 90.000,E1 103.647} C_DIS
LIN {X -0.001,Y -596.837,Z 511.371,A 0.000,B 0.000,C 90.000,E1 102.715} C_DIS
LIN {X 0.187,Y -603.705,Z 511.367,A 0.000,B 0.000,C 90.000,E1 101.951} C_DIS
LIN {X 0.187,Y -609.333,Z 511.363,A 0.000,B 0.000,C 90.000,E1 101.299} C_DIS
LIN {X -0.264,Y -612.401,Z 511.361,A 0.000,B 0.000,C 90.000,E1 100.950} C_DIS
LIN {X -0.096,Y -615.582,Z 511.359,A 0.000,B 0.000,C 90.000,E1 100.546} C_DIS
LIN {X 0.275,Y -623.064,Z 511.353,A 0.000,B 0.000,C 90.000,E1 99.500} C_DIS
LIN {X 0.137,Y -628.155,Z 511.349,A 0.000,B 0.000,C 90.000,E1 98.746} C_DIS
LIN {X 0.192,Y -632.083,Z 511.345,A 0.000,B 0.000,C 90.000,E1 98.106} C_DIS
LIN {X 0.137,Y -636.375,Z 511.341,A 0.000,B 0.000,C 90.000,E1 97.352} C_DIS
LIN {X 0.176,Y -639.757,Z 511.337,A 0.000,B 0.000,C 90.000,E1 96.720} C_DIS
LIN {X -0.140,Y -641.713,Z 511.335,A 0.000,B 0.000,C 90.000,E1 96.372} C_DIS
LIN {X 0.285,Y -646.368,Z 511.330,A 0.000,B 0.000,C 90.000,E1 95.334} C_DIS
LIN {X 0.291,Y -649.769,Z 511.326,A 0.000,B 0.000,C 90.000,E1 94.588} C_DIS
LIN {X 0.331,Y -652.750,Z 511.322,A 0.000,B 0.000,C 90.000,E1 93.841} C_DIS
LIN {X -0.087,Y -654.561,Z 511.319,A 0.000,B 0.000,C 90.000,E1 93.383} C_DIS
LIN {X 0.198,Y -656.173,Z 511.316,A 0.000,B 0.000,C 90.000,E1 92.865} C_DIS
LIN {X -0.195,Y -657.615,Z 511.313,A 0.000,B 0.000,C 90.000,E1 92.407} C_DIS
LIN {X -0.085,Y -659.361,Z 511.309,A 0.000,B 0.000,C 90.000,E1 91.661} C_DIS
LIN {X 0.204,Y -660.241,Z 511.307,A 0.000,B 0.000,C 90.000,E1 91.146} C_DIS
LIN {X -0.159,Y -660.928,Z 511.304,A 0.000,B 0.000,C 90.000,E1 90.688} C_DIS
LIN {X 0.145,Y -661.335,Z 511.301,A 0.000,B 0.000,C 90.000,E1 90.172} C_DIS
LIN {X 0.275,Y -661.481,Z 511.297,A 0.000,B 0.000,C 90.000,E1 89.427} C_DIS
LIN {X -0.078,Y -661.374,Z 511.294,A 0.000,B 0.000,C 90.000,E1 88.969} C_DIS
LIN {X 0.227,Y -661.097,Z 511.292,A 0.000,B 0.000,C 90.000,E1 88.453} C_DIS
LIN {X -0.288,Y -660.233,Z 511.287,A 0.000,B 0.000,C 90.000,E1 87.764} C_DIS
LIN {X 0.007,Y -659.477,Z 511.285,A 0.000,B 0.000,C 90.000,E1 87.249} C_DIS
LIN {X 0.143,Y -657.996,Z 511.281,A 0.000,B 0.000,C 90.000,E1 86.502} C_DIS
LIN {X -0.241,Y -656.830,Z 511.278,A 0.000,B 0.000,C 90.000,E1 86.045} C_DIS
LIN {X 0.070,Y -655.458,Z 511.275,A 0.000,B 0.000,C 90.000,E1 85.527} C_DIS
LIN {X -0.280,Y -653.923,Z 511.272,A 0.000,B 0.000,C 90.000,E1 85.065} C_DIS
LIN {X -0.197,Y -651.159,Z 511.268,A 0.000,B 0.000,C 90.000,E1 84.318} C_DIS
LIN {X -0.146,Y -648.002,Z 511.264,A 0.000,B 0.000,C 90.000,E1 83.571} C_DIS
LIN {X -0.052,Y -644.629,Z 511.260,A 0.000,B 0.000,C 90.000,E1 82.818} C_DIS
LIN {X 0.302,Y -642.790,Z 511.258,A 0.000,B 0.000,C 90.000,E1 82.413} C_DIS
LIN {X 0.342,Y -638.782,Z 511.254,A 0.000,B 0.000,C 90.000,E1 81.659} C_DIS
LIN {X -0.106,Y -635.941,Z 511.251,A 0.000,B 0.000,C 90.000,E1 81.197} C_DIS
LIN {X 0.013,Y -632.223,Z 511.248,A 0.000,B 0.000,C 90.000,E1 80.557} C_DIS
LIN {X -0.053,Y -627.258,Z 511.243,A 0.000,B 0.000,C 90.000,E1 79.803} C_DIS
LIN {X -0.223,Y -621.035,Z 511.238,A 0.000,B 0.000,C 90.000,E1 78.926} C_DIS
LIN {X 0.235,Y -615.245,Z 511.234,A 0.000,B 0.000,C 90.000,E1 78.117} C_DIS
LIN {X -0.240,Y -611.055,Z 511.231,A 0.000,B 0.000,C 90.000,E1 77.645} C_DIS
LIN {X -0.203,Y -605.188,Z 511.228,A 0.000,B 0.000,C 90.000,E1 76.992} C_DIS
LIN {X -0.076,Y -600.129,Z 511.225,A 0.000,B 0.000,C 90.000,E1 76.464} C_DIS
LIN {X 0.177,Y -594.774,Z 511.222,A 0.000,B 0.000,C 90.000,E1 75.936} C_DIS
LIN {X 0.002,Y -589.215,Z 511.219,A 0.000,B 0.000,C 90.000,E1 75.463} C_DIS
LIN {X 0.074,Y -583.370,Z 511.217,A 0.000,B 0.000,C 90.000,E1 74.991} C_DIS
LIN {X -0.199,Y -578.708,Z 511.215,A 0.000,B 0.000,C 90.000,E1 74.685} C_DIS
LIN {X -0.120,Y -572.463,Z 511.213,A 0.000,B 0.000,C 90.000,E1 74.267} C_DIS
LIN {X 0.128,Y -565.794,Z 511.210,A 0.000,B 0.000,C 90.000,E1 73.866} C_DIS
LIN {X 0.156,Y -561.033,Z 511.209,A 0.000,B 0.000,C 90.000,E1 73.614} C_DIS
LIN {X -0.185,Y -553.951,Z 511.207,A 0.000,B 0.000,C 90.000,E1 73.323} C_DIS
LIN {X 0.040,Y -546.452,Z 511.206,A 0.000,B 0.000,C 90.000,E1 73.015} C_DIS
LIN {X 0.006,Y -540.996,Z 511.205,A 0.000,B 0.000,C 90.000,E1 72.834} C_DIS
LIN {X 0.216,Y -533.231,Z 511.203,A 0.000,B 0.000,C 90.000,E1 72.598} C_DIS
LIN {X -0.076,Y -527.222,Z 511.203,A 0.000,B 0.000,C 90.000,E1 72.489} C_DIS
LIN {X 0.189,Y -519.290,Z 511.202,A 0.000,B 0.000,C 90.000,E1 72.308} C_DIS
LIN {X -0.069,Y -502.103,Z 511.200,A 0.000,B 0.000,C 90.000,E1 72.054} C_DIS
LIN {X -0.108,Y -493.633,Z 511.200,A 0.000,B 0.000,C 90.000,E1 71.945} C_DIS
LIN {X 0.130,Y -473.792,Z 511.199,A 0.000,B 0.000,C 90.000,E1 71.710} C_DIS
LIN {X 0.082,Y -473.479,Z 511.198,A 0.000,B 0.000,C 90.000,E1 71.710} C_DIS
LIN {X -0.044,Y -465.456,Z 511.172,A 0.000,B 0.000,C 90.000,E1 66.975} C_DIS
LIN {X 0.143,Y -457.022,Z 511.149,A 0.000,B 0.000,C 90.000,E1 62.820} C_DIS
LIN {X -0.155,Y -455.433,Z 511.144,A 0.000,B 0.000,C 90.000,E1 61.897} C_DIS
LIN {X -0.211,Y -447.715,Z 511.125,A 0.000,B 0.000,C 90.000,E1 58.535} C_DIS
LIN {X -0.251,Y -447.720,Z 511.125,A 0.000,B 0.000,C 90.000,E1 58.535} C_DIS
LIN {X 0.168,Y -450.847,Z 511.121,A 0.000,B 0.000,C 90.000,E1 57.661} C_DIS
LIN {X 0.042,Y -454.186,Z 511.115,A 0.000,B 0.000,C 90.000,E1 56.707} C_DIS
LIN {X -0.148,Y -456.270,Z 511.112,A 0.000,B 0.000,C 90.000,E1 56.087} C_DIS
LIN {X 0.153,Y -460.114,Z 511.104,A 0.000,B 0.000,C 90.000,E1 54.769} C_DIS
LIN {X 0.138,Y -463.173,Z 511.097,A 0.000,B 0.000,C 90.000,E1 53.497} C_DIS
LIN {X -0.114,Y -463.916,Z 511.096,A 0.000,B 0.000,C 90.000,E1 53.210} C_DIS
LIN {X -0.205,Y -465.683,Z 511.090,A 0.000,B 0.000,C 90.000,E1 52.271} C_DIS
LIN {X 0.017,Y -467.215,Z 511.085,A 0.000,B 0.000,C 90.000,E1 51.295} C_DIS
LIN {X 0.032,Y -468.947,Z 511.078,A 0.000,B 0.000,C 90.000,E1 50.033} C_DIS
LIN {X 0.068,Y -470.452,Z 511.071,A 0.000,B 0.000,C 90.000,E1 48.771} C_DIS
LIN {X -0.234,Y -471.593,Z 511.064,A 0.000,B 0.000,C 90.000,E1 47.553} C_DIS
LIN {X 0.031,Y -472.303,Z 511.059,A 0.000,B 0.000,C 90.000,E1 46.581} C_DIS
LIN {X 0.075,Y -473.048,Z 511.052,A 0.000,B 0.000,C 90.000,E1 45.324} C_DIS
LIN {X 0.267,Y -473.324,Z 511.048,A 0.000,B 0.000,C 90.000,E1 44.676} C_DIS
LIN {X -0.114,Y -473.622,Z 511.043,A 0.000,B 0.000,C 90.000,E1 43.785} C_DIS
LIN {X -0.054,Y -473.715,Z 511.036,A 0.000,B 0.000,C 90.000,E1 42.528} C_DIS
LIN {X 0.004,Y -473.581,Z 511.029,A 0.000,B 0.000,C 90.000,E1 41.272} C_DIS
LIN {X 0.101,Y -473.233,Z 511.022,A 0.000,B 0.000,C 90.000,E1 40.011} C_DIS
LIN {X -0.021,Y -472.613,Z 511.014,A 0.000,B 0.000,C 90.000,E1 38.463} C_DIS
LIN {X 0.217,Y -471.790,Z 511.005,A 0.000,B 0.000,C 90.000,E1 36.870} C_DIS
LIN {X 0.155,Y -470.934,Z 510.996,A 0.000,B 0.000,C 90.000,E1 35.311} C_DIS
LIN {X -0.129,Y -470.327,Z 510.991,A 0.000,B 0.000,C 90.000,E1 34.405} C_DIS
LIN {X -0.097,Y -469.269,Z 510.982,A 0.000,B 0.000,C 90.000,E1 32.832} C_DIS
LIN {X 0.152,Y -468.363,Z 510.975,A 0.000,B 0.000,C 90.000,E1 31.544} C_DIS
LIN {X 0.048,Y -466.848,Z 510.965,A 0.000,B 0.000,C 90.000,E1 29.667} C_DIS
LIN {X 0.078,Y -465.304,Z 510.954,A 0.000,B 0.000,C 90.000,E1 27.769} C_DIS
LIN {X 0.136,Y -464.109,Z 510.946,A 0.000,B 0.000,C 90.000,E1 26.181} C_DIS
LIN {X 0.223,Y -462.565,Z 510.933,A 0.000,B 0.000,C 90.000,E1 23.951} C_DIS
LIN {X 0.155,Y -460.949,Z 510.917,A 0.000,B 0.000,C 90.000,E1 21.099} C_DIS
LIN {X -0.131,Y -459.975,Z 510.905,A 0.000,B 0.000,C 90.000,E1 18.906} C_DIS
LIN {X 0.187,Y -459.031,Z 510.891,A 0.000,B 0.000,C 90.000,E1 16.315} C_DIS
LIN {X 0.097,Y -458.454,Z 510.877,A 0.000,B 0.000,C 90.000,E1 13.772} C_DIS
LIN {X 0.106,Y -458.416,Z 510.864,A 0.000,B 0.000,C 90.000,E1 11.535} C_DIS
LIN {X -0.063,Y -458.796,Z 510.848,A 0.000,B 0.000,C 90.000,E1 8.681} C_DIS
LIN {X -0.238,Y -459.808,Z 510.831,A 0.000,B 0.000,C 90.000,E1 5.511} C_DIS
LIN {X 0.114,Y -460.791,Z 510.820,A 0.000,B 0.000,C 90.000,E1 3.555} C_DIS
LIN {X -0.009,Y -462.088,Z 510.809,A 0.000,B 0.000,C 90.000,E1 1.661} C_DIS
LIN {X 0.175,Y -463.578,Z 510.799,A 0.000,B 0.000,C 90.000,E1 359.771} C_DIS
LIN {X -0.139,Y -465.786,Z 510.787,A 0.000,B 0.000,C 90.000,E1 357.593} C_DIS
LIN {X -0.112,Y -468.797,Z 510.773,A 0.000,B 0.000,C 90.000,E1 355.065} C_DIS
LIN {X 0.181,Y -470.814,Z 510.764,A 0.000,B 0.000,C 90.000,E1 353.457} C_DIS
LIN {X 0.150,Y -472.846,Z 510.755,A 0.000,B 0.000,C 90.000,E1 351.894} C_DIS
LIN {X 0.163,Y -475.002,Z 510.746,A 0.000,B 0.000,C 90.000,E1 350.330} C_DIS
LIN {X -0.016,Y -478.282,Z 510.734,A 0.000,B 0.000,C 90.000,E1 348.173} C_DIS
LIN {X 0.117,Y -484.835,Z 510.714,A 0.000,B 0.000,C 90.000,E1 344.448} C_DIS
LIN {X 0.197,Y -488.544,Z 510.703,A 0.000,B 0.000,C 90.000,E1 342.598} C_DIS
LIN {X 0.040,Y -492.406,Z 510.693,A 0.000,B 0.000,C 90.000,E1 340.786} C_DIS
LIN {X 0.134,Y -496.224,Z 510.683,A 0.000,B 0.000,C 90.000,E1 338.954} C_DIS
LIN {X -0.287,Y -498.761,Z 510.677,A 0.000,B 0.000,C 90.000,E1 337.794} C_DIS
LIN {X -0.144,Y -502.463,Z 510.666,A 0.000,B 0.000,C 90.000,E1 335.973} C_DIS
LIN {X 0.003,Y -505.395,Z 510.658,A 0.000,B 0.000,C 90.000,E1 334.460} C_DIS
LIN {X -0.258,Y -508.315,Z 510.650,A 0.000,B 0.000,C 90.000,E1 332.999} C_DIS
LIN {X -0.259,Y -512.466,Z 510.638,A 0.000,B 0.000,C 90.000,E1 330.923} C_DIS
LIN {X 0.089,Y -516.701,Z 510.627,A 0.000,B 0.000,C 90.000,E1 328.820} C_DIS
LIN {X -0.075,Y -520.970,Z 510.615,A 0.000,B 0.000,C 90.000,E1 326.786} C_DIS
LIN {X -0.277,Y -525.316,Z 510.604,A 0.000,B 0.000,C 90.000,E1 324.769} C_DIS
LIN {X -0.040,Y -529.049,Z 510.594,A 0.000,B 0.000,C 90.000,E1 323.004} C_DIS
LIN {X 0.179,Y -532.702,Z 510.585,A 0.000,B 0.000,C 90.000,E1 321.251} C_DIS
LIN {X 0.074,Y -535.150,Z 510.578,A 0.000,B 0.000,C 90.000,E1 320.114} C_DIS
LIN {X 0.013,Y -538.810,Z 510.569,A 0.000,B 0.000,C 90.000,E1 318.405} C_DIS
LIN {X -0.024,Y -542.456,Z 510.559,A 0.000,B 0.000,C 90.000,E1 316.701} C_DIS
LIN {X 0.001,Y -545.997,Z 510.550,A 0.000,B 0.000,C 90.000,E1 315.000} C_DIS
LIN {X 0.102,Y -549.448,Z 510.541,A 0.000,B 0.000,C 90.000,E1 313.299} C_DIS
LIN {X -0.065,Y -553.420,Z 510.530,A 0.000,B 0.000,C 90.000,E1 311.353} C_DIS
LIN {X 0.196,Y -556.343,Z 510.522,A 0.000,B 0.000,C 90.000,E1 309.930} C_DIS
LIN {X 0.162,Y -559.358,Z 510.514,A 0.000,B 0.000,C 90.000,E1 308.543} C_DIS
LIN {X 0.184,Y -562.204,Z 510.507,A 0.000,B 0.000,C 90.000,E1 307.156} C_DIS
LIN {X 0.133,Y -566.034,Z 510.496,A 0.000,B 0.000,C 90.000,E1 305.231} C_DIS
LIN {X 0.311,Y -570.006,Z 510.485,A 0.000,B 0.000,C 90.000,E1 303.293} C_DIS
LIN {X 0.144,Y -573.483,Z 510.476,A 0.000,B 0.000,C 90.000,E1 301.671} C_DIS
LIN {X -0.089,Y -576.236,Z 510.469,A 0.000,B 0.000,C 90.000,E1 300.335} C_DIS
LIN {X 0.224,Y -579.014,Z 510.461,A 0.000,B 0.000,C 90.000,E1 298.949} C_DIS
LIN {X -0.206,Y -581.840,Z 510.453,A 0.000,B 0.000,C 90.000,E1 297.641} C_DIS
LIN {X -0.085,Y -583.292,Z 510.449,A 0.000,B 0.000,C 90.000,E1 296.821} C_DIS
LIN {X 0.317,Y -584.400,Z 510.445,A 0.000,B 0.000,C 90.000,E1 295.976} C_DIS
LIN {X 0.067,Y -584.947,Z 510.442,A 0.000,B 0.000,C 90.000,E1 295.463} C_DIS
LIN {X -0.057,Y -585.130,Z 510.440,A 0.000,B 0.000,C 90.000,E1 295.207} C_DIS
LIN {X -0.182,Y -585.152,Z 510.439,A 0.000,B 0.000,C 90.000,E1 294.951} C_DIS
LIN {X 0.226,Y -585.341,Z 510.437,A 0.000,B 0.000,C 90.000,E1 294.643} C_DIS
LIN {X -0.145,Y -585.239,Z 510.433,A 0.000,B 0.000,C 90.000,E1 293.875} C_DIS
LIN {X -0.094,Y -585.065,Z 510.430,A 0.000,B 0.000,C 90.000,E1 293.334} C_DIS
LIN {X -0.002,Y -585.501,Z 510.421,A 0.000,B 0.000,C 90.000,E1 291.716} C_DIS
LIN {X 0.016,Y -586.315,Z 510.413,A 0.000,B 0.000,C 90.000,E1 290.375} C_DIS
LIN {X -0.036,Y -586.656,Z 510.409,A 0.000,B 0.000,C 90.000,E1 289.577} C_DIS
LIN {X -0.004,Y -587.036,Z 510.401,A 0.000,B 0.000,C 90.000,E1 288.236} C_DIS
LIN {X -0.156,Y -587.151,Z 510.394,A 0.000,B 0.000,C 90.000,E1 286.913} C_DIS
LIN {X -0.152,Y -587.108,Z 510.388,A 0.000,B 0.000,C 90.000,E1 285.843} C_DIS
LIN {X -0.219,Y -587.051,Z 510.379,A 0.000,B 0.000,C 90.000,E1 284.245} C_DIS
LIN {X -0.040,Y -586.832,Z 510.369,A 0.000,B 0.000,C 90.000,E1 282.355} C_DIS
LIN {X 0.066,Y -586.631,Z 510.361,A 0.000,B 0.000,C 90.000,E1 281.007} C_DIS
LIN {X -0.122,Y -586.257,Z 510.351,A 0.000,B 0.000,C 90.000,E1 279.151} C_DIS
LIN {X -0.138,Y -585.903,Z 510.343,A 0.000,B 0.000,C 90.000,E1 277.814} C_DIS
LIN {X -0.080,Y -585.339,Z 510.334,A 0.000,B 0.000,C 90.000,E1 276.201} C_DIS
LIN {X 0.150,Y -584.821,Z 510.328,A 0.000,B 0.000,C 90.000,E1 275.106} C_DIS
LIN {X -0.042,Y -583.981,Z 510.321,A 0.000,B 0.000,C 90.000,E1 273.784} C_DIS
LIN {X -0.287,Y -582.964,Z 510.314,A 0.000,B 0.000,C 90.000,E1 272.465} C_DIS
LIN {X 0.208,Y -581.438,Z 510.305,A 0.000,B 0.000,C 90.000,E1 270.802} C_DIS
LIN {X -0.094,Y -579.964,Z 510.297,A 0.000,B 0.000,C 90.000,E1 269.484} C_DIS
LIN {X -0.008,Y -578.753,Z 510.291,A 0.000,B 0.000,C 90.000,E1 268.396} C_DIS
LIN {X -0.160,Y -576.828,Z 510.282,A 0.000,B 0.000,C 90.000,E1 266.788} C_DIS
LIN {X -0.284,Y -575.850,Z 510.278,A 0.000,B 0.000,C 90.000,E1 265.988} C_DIS
LIN {X 0.126,Y -573.796,Z 510.269,A 0.000,B 0.000,C 90.000,E1 264.318} C_DIS
LIN {X -0.074,Y -571.464,Z 510.259,A 0.000,B 0.000,C 90.000,E1 262.704} C_DIS
LIN {X 0.128,Y -569.343,Z 510.252,A 0.000,B 0.000,C 90.000,E1 261.319} C_DIS
LIN {X -0.010,Y -566.782,Z 510.243,A 0.000,B 0.000,C 90.000,E1 259.690} C_DIS
LIN {X 0.297,Y -564.579,Z 510.235,A 0.000,B 0.000,C 90.000,E1 258.285} C_DIS
LIN {X 0.173,Y -561.775,Z 510.226,A 0.000,B 0.000,C 90.000,E1 256.645} C_DIS
LIN {X -0.174,Y -559.817,Z 510.220,A 0.000,B 0.000,C 90.000,E1 255.574} C_DIS
LIN {X -0.001,Y -557.663,Z 510.214,A 0.000,B 0.000,C 90.000,E1 254.448} C_DIS
LIN {X 0.134,Y -555.388,Z 510.207,A 0.000,B 0.000,C 90.000,E1 253.323} C_DIS
LIN {X 0.242,Y -551.720,Z 510.198,A 0.000,B 0.000,C 90.000,E1 251.638} C_DIS
LIN {X 0.186,Y -548.428,Z 510.190,A 0.000,B 0.000,C 90.000,E1 250.242} C_DIS
LIN {X -0.194,Y -544.158,Z 510.181,A 0.000,B 0.000,C 90.000,E1 248.592} C_DIS
LIN {X -0.200,Y -540.434,Z 510.173,A 0.000,B 0.000,C 90.000,E1 247.177} C_DIS
LIN {X -0.285,Y -537.282,Z 510.167,A 0.000,B 0.000,C 90.000,E1 246.049} C_DIS
LIN {X 0.294,Y -533.999,Z 510.160,A 0.000,B 0.000,C 90.000,E1 244.845} C_DIS
LIN {X 0.056,Y -529.798,Z 510.152,A 0.000,B 0.000,C 90.000,E1 243.435} C_DIS
LIN {X 0.208,Y -525.431,Z 510.144,A 0.000,B 0.000,C 90.000,E1 241.975} C_DIS
LIN {X 0.054,Y -521.046,Z 510.136,A 0.000,B 0.000,C 90.000,E1 240.539} C_DIS
LIN {X 0.078,Y -516.629,Z 510.128,A 0.000,B 0.000,C 90.000,E1 239.076} C_DIS
LIN {X 0.291,Y -512.004,Z 510.120,A 0.000,B 0.000,C 90.000,E1 237.582} C_DIS
LIN {X 0.089,Y -508.245,Z 510.114,A 0.000,B 0.000,C 90.000,E1 236.421} C_DIS
LIN {X 0.089,Y -500.601,Z 510.100,A 0.000,B 0.000,C 90.000,E1 234.036} C_DIS
LIN {X 0.173,Y -491.695,Z 510.084,A 0.000,B 0.000,C 90.000,E1 231.009} C_DIS
LIN {X -0.179,Y -484.936,Z 510.070,A 0.000,B 0.000,C 90.000,E1 228.609} C_DIS
LIN {X -0.011,Y -480.109,Z 510.060,A 0.000,B 0.000,C 90.000,E1 226.743} C_DIS
LIN {X 0.032,Y -475.240,Z 510.049,A 0.000,B 0.000,C 90.000,E1 224.879} C_DIS
LIN {X -0.124,Y -471.322,Z 510.041,A 0.000,B 0.000,C 90.000,E1 223.338} C_DIS
LIN {X 0.046,Y -466.839,Z 510.030,A 0.000,B 0.000,C 90.000,E1 221.434} C_DIS
LIN {X -0.012,Y -461.115,Z 510.016,A 0.000,B 0.000,C 90.000,E1 218.910} C_DIS
LIN {X 0.006,Y -456.953,Z 510.006,A 0.000,B 0.000,C 90.000,E1 216.996} C_DIS
LIN {X 0.183,Y -451.626,Z 509.991,A 0.000,B 0.000,C 90.000,E1 214.405} C_DIS
LIN {X 0.247,Y -447.222,Z 509.979,A 0.000,B 0.000,C 90.000,E1 212.133} C_DIS
LIN {X 0.040,Y -443.605,Z 509.968,A 0.000,B 0.000,C 90.000,E1 210.207} C_DIS
LIN {X 0.176,Y -439.491,Z 509.955,A 0.000,B 0.000,C 90.000,E1 207.897} C_DIS
LIN {X -0.070,Y -436.588,Z 509.946,A 0.000,B 0.000,C 90.000,E1 206.283} C_DIS
LIN {X 0.050,Y -433.170,Z 509.935,A 0.000,B 0.000,C 90.000,E1 204.283} C_DIS
LIN {X 0.100,Y -429.846,Z 509.924,A 0.000,B 0.000,C 90.000,E1 202.280} C_DIS
LIN {X -0.102,Y -425.746,Z 509.909,A 0.000,B 0.000,C 90.000,E1 199.631} C_DIS
LIN {X 0.073,Y -422.013,Z 509.894,A 0.000,B 0.000,C 90.000,E1 196.913} C_DIS
LIN {X -0.041,Y -419.459,Z 509.883,A 0.000,B 0.000,C 90.000,E1 194.898} C_DIS
LIN {X -0.159,Y -416.622,Z 509.870,A 0.000,B 0.000,C 90.000,E1 192.535} C_DIS
LIN {X -0.128,Y -414.008,Z 509.856,A 0.000,B 0.000,C 90.000,E1 190.141} C_DIS
LIN {X 0.159,Y -411.516,Z 509.843,A 0.000,B 0.000,C 90.000,E1 187.701} C_DIS
LIN {X -0.172,Y -409.389,Z 509.831,A 0.000,B 0.000,C 90.000,E1 185.682} C_DIS
LIN {X 0.137,Y -405.938,Z 509.810,A 0.000,B 0.000,C 90.000,E1 181.835} C_DIS
LIN {X 0.026,Y -404.791,Z 509.801,A 0.000,B 0.000,C 90.000,E1 180.115} C_DIS
LIN {X 0.200,Y -403.283,Z 509.785,A 0.000,B 0.000,C 90.000,E1 177.306} C_DIS
LIN {X -0.063,Y -402.276,Z 509.766,A 0.000,B 0.000,C 90.000,E1 173.856} C_DIS
LIN {X 0.175,Y -402.147,Z 509.746,A 0.000,B 0.000,C 90.000,E1 170.330} C_DIS
LIN {X -0.189,Y -402.540,Z 509.731,A 0.000,B 0.000,C 90.000,E1 167.589} C_DIS
LIN {X 0.211,Y -403.457,Z 509.714,A 0.000,B 0.000,C 90.000,E1 164.393} C_DIS
LIN {X -0.204,Y -404.374,Z 509.702,A 0.000,B 0.000,C 90.000,E1 162.362} C_DIS
LIN {X 0.140,Y -405.791,Z 509.688,A 0.000,B 0.000,C 90.000,E1 159.880} C_DIS
LIN {X 0.164,Y -407.681,Z 509.673,A 0.000,B 0.000,C 90.000,E1 157.102} C_DIS
LIN {X -0.092,Y -409.060,Z 509.663,A 0.000,B 0.000,C 90.000,E1 155.409} C_DIS
LIN {X -0.063,Y -410.270,Z 509.656,A 0.000,B 0.000,C 90.000,E1 154.024} C_DIS
LIN {X 0.086,Y -411.663,Z 509.646,A 0.000,B 0.000,C 90.000,E1 152.281} C_DIS
LIN {X -0.031,Y -412.774,Z 509.638,A 0.000,B 0.000,C 90.000,E1 150.923} C_DIS
LIN {X 0.003,Y -414.067,Z 509.629,A 0.000,B 0.000,C 90.000,E1 149.203} C_DIS
LIN {X -0.074,Y -415.281,Z 509.619,A 0.000,B 0.000,C 90.000,E1 147.502} C_DIS
LIN {X -0.125,Y -416.391,Z 509.610,A 0.000,B 0.000,C 90.000,E1 145.801} C_DIS
LIN {X -0.139,Y -417.840,Z 509.597,A 0.000,B 0.000,C 90.000,E1 143.417} C_DIS
LIN {X -0.013,Y -418.771,Z 509.587,A 0.000,B 0.000,C 90.000,E1 141.698} C_DIS
LIN {X 0.062,Y -419.610,Z 509.578,A 0.000,B 0.000,C 90.000,E1 139.989} C_DIS
LIN {X -0.166,Y -420.273,Z 509.568,A 0.000,B 0.000,C 90.000,E1 138.324} C_DIS
LIN {X 0.005,Y -420.704,Z 509.561,A 0.000,B 0.000,C 90.000,E1 136.944} C_DIS
LIN {X 0.059,Y -420.952,Z 509.551,A 0.000,B 0.000,C 90.000,E1 135.243} C_DIS
LIN {X -0.260,Y -421.037,Z 509.546,A 0.000,B 0.000,C 90.000,E1 134.271} C_DIS
LIN {X 0.211,Y -420.832,Z 509.538,A 0.000,B 0.000,C 90.000,E1 132.852} C_DIS
LIN {X 0.193,Y -420.558,Z 509.533,A 0.000,B 0.000,C 90.000,E1 131.838} C_DIS
LIN {X -0.223,Y -419.720,Z 509.525,A 0.000,B 0.000,C 90.000,E1 130.539} C_DIS
LIN {X 0.058,Y -418.977,Z 509.519,A 0.000,B 0.000,C 90.000,E1 129.483} C_DIS
LIN {X 0.059,Y -417.328,Z 509.508,A 0.000,B 0.000,C 90.000,E1 127.443} C_DIS
LIN {X 0.011,Y -415.944,Z 509.499,A 0.000,B 0.000,C 90.000,E1 125.804} C_DIS
LIN {X -0.027,Y -415.949,Z 509.499,A 0.000,B 0.000,C 90.000,E1 125.804} C_DIS
LIN {X 0.054,Y -425.589,Z 509.478,A 0.000,B 0.000,C 90.000,E1 122.005} C_DIS
LIN {X -0.002,Y -430.624,Z 509.469,A 0.000,B 0.000,C 90.000,E1 120.335} C_DIS
LIN {X -0.009,Y -441.528,Z 509.445,A 0.000,B 0.000,C 90.000,E1 116.027} C_DIS
LIN {X 0.119,Y -444.445,Z 509.439,A 0.000,B 0.000,C 90.000,E1 115.027} C_DIS
LIN {X 0.017,Y -445.918,Z 509.436,A 0.000,B 0.000,C 90.000,E1 114.387} C_DIS
LIN {X 0.155,Y -455.324,Z 509.414,A 0.000,B 0.000,C 90.000,E1 110.482} C_DIS
LIN {X -0.050,Y -457.124,Z 509.410,A 0.000,B 0.000,C 90.000,E1 109.866} C_DIS
LIN {X -0.125,Y -458.743,Z 509.406,A 0.000,B 0.000,C 90.000,E1 109.014} C_DIS
LIN {X 0.269,Y -458.836,Z 509.406,A 0.000,B 0.000,C 90.000,E1 108.960} C_DIS
LIN {X -0.043,Y -472.659,Z 509.403,A 0.000,B 0.000,C 90.000,E1 108.598} C_DIS
LIN {X 0.130,Y -490.547,Z 509.400,A 0.000,B 0.000,C 90.000,E1 108.055} C_DIS
LIN {X -0.119,Y -504.581,Z 509.398,A 0.000,B 0.000,C 90.000,E1 107.638} C_DIS
LIN {X 0.038,Y -518.556,Z 509.395,A 0.000,B 0.000,C 90.000,E1 107.149} C_DIS
LIN {X 0.006,Y -525.352,Z 509.394,A 0.000,B 0.000,C 90.000,E1 106.913} C_DIS
LIN {X -0.201,Y -535.709,Z 509.392,A 0.000,B 0.000,C 90.000,E1 106.551} C_DIS
LIN {X 0.025,Y -542.249,Z 509.390,A 0.000,B 0.000,C 90.000,E1 106.260} C_DIS
LIN {X -0.072,Y -550.414,Z 509.388,A 0.000,B 0.000,C 90.000,E1 105.898} C_DIS
LIN {X 0.240,Y -552.094,Z 509.388,A 0.000,B 0.000,C 90.000,E1 105.788} C_DIS
LIN {X -0.228,Y -556.319,Z 509.387,A 0.000,B 0.000,C 90.000,E1 105.607} C_DIS
LIN {X 0.134,Y -558.215,Z 509.386,A 0.000,B 0.000,C 90.000,E1 105.481} C_DIS
LIN {X -0.294,Y -564.133,Z 509.384,A 0.000,B 0.000,C 90.000,E1 105.190} C_DIS
LIN {X 0.008,Y -570.165,Z 509.382,A 0.000,B 0.000,C 90.000,E1 104.773} C_DIS
LIN {X -0.004,Y -576.131,Z 509.380,A 0.000,B 0.000,C 90.000,E1 104.356} C_DIS
LIN {X 0.265,Y -578.766,Z 509.379,A 0.000,B 0.000,C 90.000,E1 104.120} C_DIS
LIN {X 0.096,Y -581.331,Z 509.378,A 0.000,B 0.000,C 90.000,E1 103.953} C_DIS
LIN {X -0.270,Y -586.811,Z 509.375,A 0.000,B 0.000,C 90.000,E1 103.536} C_DIS
LIN {X -0.216,Y -590.553,Z 509.373,A 0.000,B 0.000,C 90.000,E1 103.175} C_DIS
LIN {X 0.247,Y -593.251,Z 509.372,A 0.000,B 0.000,C 90.000,E1 102.883} C_DIS
LIN {X -0.067,Y -597.765,Z 509.369,A 0.000,B 0.000,C 90.000,E1 102.479} C_DIS
LIN {X -0.001,Y -603.785,Z 509.366,A 0.000,B 0.000,C 90.000,E1 101.827} C_DIS
LIN {X -0.148,Y -609.530,Z 509.362,A 0.000,B 0.000,C 90.000,E1 101.186} C_DIS
LIN {X -0.248,Y -614.948,Z 509.359,A 0.000,B 0.000,C 90.000,E1 100.546} C_DIS
LIN {X 0.077,Y -621.850,Z 509.353,A 0.000,B 0.000,C 90.000,E1 99.613} C_DIS
LIN {X 0.140,Y -625.405,Z 509.351,A 0.000,B 0.000,C 90.000,E1 99.095} C_DIS
LIN {X 0.328,Y -628.799,Z 509.348,A 0.000,B 0.000,C 90.000,E1 98.568} C_DIS
LIN {X -0.328,Y -632.774,Z 509.344,A 0.000,B 0.000,C 90.000,E1 97.992} C_DIS
LIN {X -0.240,Y -636.352,Z 509.341,A 0.000,B 0.000,C 90.000,E1 97.352} C_DIS
LIN {X -0.205,Y -639.833,Z 509.337,A 0.000,B 0.000,C 90.000,E1 96.720} C_DIS
LIN {X -0.134,Y -643.023,Z 509.334,A 0.000,B 0.000,C 90.000,E1 96.087} C_DIS
LIN {X 0.197,Y -648.267,Z 509.328,A 0.000,B 0.000,C 90.000,E1 94.935} C_DIS
LIN {X -0.202,Y -650.458,Z 509.325,A 0.000,B 0.000,C 90.000,E1 94.473} C_DIS
LIN {X -0.156,Y -653.474,Z 509.321,A 0.000,B 0.000,C 90.000,E1 93.726} C_DIS
LIN {X -0.082,Y -656.061,Z 509.317,A 0.000,B 0.000,C 90.000,E1 92.980} C_DIS
LIN {X -0.013,Y -658.183,Z 509.312,A 0.000,B 0.000,C 90.000,E1 92.236} C_DIS
LIN {X 0.290,Y -659.366,Z 509.310,A 0.000,B 0.000,C 90.000,E1 91.718} C_DIS
LIN {X -0.081,Y -660.337,Z 509.307,A 0.000,B 0.000,C 90.000,E1 91.260} C_DIS
LIN {X 0.038,Y -661.241,Z 509.303,A 0.000,B 0.000,C 90.000,E1 90.516} C_DIS
LIN {X -0.318,Y -661.599,Z 509.300,A 0.000,B 0.000,C 90.000,E1 90.057} C_DIS
LIN {X -0.184,Y -661.601,Z 509.296,A 0.000,B 0.000,C 90.000,E1 89.312} C_DIS
LIN {X 0.123,Y -661.397,Z 509.293,A 0.000,B 0.000,C 90.000,E1 88.797} C_DIS
LIN {X -0.232,Y -661.039,Z 509.291,A 0.000,B 0.000,C 90.000,E1 88.339} C_DIS
LIN {X 0.093,Y -660.465,Z 509.288,A 0.000,B 0.000,C 90.000,E1 87.822} C_DIS
LIN {X 0.206,Y -659.147,Z 509.284,A 0.000,B 0.000,C 90.000,E1 87.078} C_DIS
LIN {X -0.319,Y -657.612,Z 509.280,A 0.000,B 0.000,C 90.000,E1 86.388} C_DIS
LIN {X -0.200,Y -655.535,Z 509.276,A 0.000,B 0.000,C 90.000,E1 85.641} C_DIS
LIN {X -0.100,Y -653.070,Z 509.272,A 0.000,B 0.000,C 90.000,E1 84.894} C_DIS
LIN {X 0.188,Y -651.204,Z 509.269,A 0.000,B 0.000,C 90.000,E1 84.375} C_DIS
LIN {X 0.082,Y -646.938,Z 509.263,A 0.000,B 0.000,C 90.000,E1 83.394} C_DIS
LIN {X 0.086,Y -643.400,Z 509.259,A 0.000,B 0.000,C 90.000,E1 82.648} C_DIS
LIN {X -0.002,Y -638.669,Z 509.254,A 0.000,B 0.000,C 90.000,E1 81.781} C_DIS
LIN {X 0.273,Y -635.803,Z 509.252,A 0.000,B 0.000,C 90.000,E1 81.254} C_DIS
LIN {X -0.193,Y -632.786,Z 509.249,A 0.000,B 0.000,C 90.000,E1 80.792} C_DIS
LIN {X -0.255,Y -627.739,Z 509.245,A 0.000,B 0.000,C 90.000,E1 80.038} C_DIS
LIN {X -0.206,Y -623.194,Z 509.241,A 0.000,B 0.000,C 90.000,E1 79.398} C_DIS
LIN {X 0.188,Y -619.577,Z 509.238,A 0.000,B 0.000,C 90.000,E1 78.870} C_DIS
LIN {X -0.193,Y -615.780,Z 509.236,A 0.000,B 0.000,C 90.000,E1 78.409} C_DIS
LIN {X -0.121,Y -610.428,Z 509.232,A 0.000,B 0.000,C 90.000,E1 77.757} C_DIS
LIN {X -0.114,Y -604.529,Z 509.228,A 0.000,B 0.000,C 90.000,E1 77.117} C_DIS
LIN {X -0.305,Y -599.635,Z 509.226,A 0.000,B 0.000,C 90.000,E1 76.645} C_DIS
LIN {X -0.049,Y -594.146,Z 509.223,A 0.000,B 0.000,C 90.000,E1 76.117} C_DIS
LIN {X -0.127,Y -588.590,Z 509.220,A 0.000,B 0.000,C 90.000,E1 75.644} C_DIS
LIN {X -0.061,Y -582.589,Z 509.218,A 0.000,B 0.000,C 90.000,E1 75.172} C_DIS
LIN {X 0.305,Y -578.011,Z 509.216,A 0.000,B 0.000,C 90.000,E1 74.810} C_DIS
LIN {X -0.104,Y -571.577,Z 509.214,A 0.000,B 0.000,C 90.000,E1 74.448} C_DIS
LIN {X -0.006,Y -566.584,Z 509.212,A 0.000,B 0.000,C 90.000,E1 74.157} C_DIS
LIN {X 0.135,Y -559.752,Z 509.210,A 0.000,B 0.000,C 90.000,E1 73.795} C_DIS
LIN {X -0.008,Y -552.567,Z 509.208,A 0.000,B 0.000,C 90.000,E1 73.504} C_DIS
LIN {X -0.194,Y -541.687,Z 509.206,A 0.000,B 0.000,C 90.000,E1 73.142} C_DIS
LIN {X -0.150,Y -529.768,Z 509.205,A 0.000,B 0.000,C 90.000,E1 72.834} C_DIS
LIN {X 0.223,Y -519.562,Z 509.204,A 0.000,B 0.000,C 90.000,E1 72.598} C_DIS
LIN {X 0.071,Y -511.182,Z 509.203,A 0.000,B 0.000,C 90.000,E1 72.489} C_DIS
LIN {X -0.162,Y -495.576,Z 509.202,A 0.000,B 0.000,C 90.000,E1 72.308} C_DIS
LIN {X -0.087,Y -484.019,Z 509.201,A 0.000,B 0.000,C 90.000,E1 72.181} C_DIS
LIN {X -0.276,Y -474.205,Z 509.201,A 0.000,B 0.000,C 90.000,E1 72.127} C_DIS
LIN {X 0.134,Y -474.165,Z 509.201,A 0.000,B 0.000,C 90.000,E1 72.072} C_DIS
LIN {X 0.081,Y -467.393,Z 509.179,A 0.000,B 0.000,C 90.000,E1 68.284} C_DIS
LIN {X -0.140,Y -465.592,Z 509.172,A 0.000,B 0.000,C 90.000,E1 67.050} C_DIS
LIN {X -0.259,Y -456.589,Z 509.148,A 0.000,B 0.000,C 90.000,E1 62.615} C_DIS
LIN {X -0.045,Y -455.549,Z 509.144,A 0.000,B 0.000,C 90.000,E1 61.948} C_DIS
LIN {X 0.210,Y -448.085,Z 509.126,A 0.000,B 0.000,C 90.000,E1 58.663} C_DIS
LIN {X 0.170,Y -448.075,Z 509.126,A 0.000,B 0.000,C 90.000,E1 58.663} C_DIS
LIN {X 0.065,Y -451.808,Z 509.121,A 0.000,B 0.000,C 90.000,E1 57.740} C_DIS
LIN {X 0.297,Y -456.357,Z 509.114,A 0.000,B 0.000,C 90.000,E1 56.421} C_DIS
LIN {X -0.145,Y -459.370,Z 509.108,A 0.000,B 0.000,C 90.000,E1 55.515} C_DIS
LIN {X 0.081,Y -461.244,Z 509.105,A 0.000,B 0.000,C 90.000,E1 54.848} C_DIS
LIN {X -0.043,Y -463.600,Z 509.100,A 0.000,B 0.000,C 90.000,E1 53.909} C_DIS
LIN {X 0.110,Y -465.068,Z 509.096,A 0.000,B 0.000,C 90.000,E1 53.256} C_DIS
LIN {X 0.038,Y -466.856,Z 509.091,A 0.000,B 0.000,C 90.000,E1 52.316} C_DIS
LIN {X -0.069,Y -467.934,Z 509.087,A 0.000,B 0.000,C 90.000,E1 51.698} C_DIS
LIN {X -0.052,Y -469.667,Z 509.080,A 0.000,B 0.000,C 90.000,E1 50.436} C_DIS
LIN {X 0.220,Y -470.843,Z 509.075,A 0.000,B 0.000,C 90.000,E1 49.461} C_DIS
LIN {X 0.153,Y -471.816,Z 509.070,A 0.000,B 0.000,C 90.000,E1 48.528} C_DIS
LIN {X -0.127,Y -472.882,Z 509.063,A 0.000,B 0.000,C 90.000,E1 47.310} C_DIS
LIN {X -0.075,Y -473.691,Z 509.056,A 0.000,B 0.000,C 90.000,E1 46.053} C_DIS
LIN {X 0.219,Y -474.181,Z 509.051,A 0.000,B 0.000,C 90.000,E1 45.081} C_DIS
LIN {X -0.052,Y -474.553,Z 509.044,A 0.000,B 0.000,C 90.000,E1 43.866} C_DIS
LIN {X -0.076,Y -474.637,Z 509.039,A 0.000,B 0.000,C 90.000,E1 42.933} C_DIS
LIN {X -0.097,Y -474.561,Z 509.033,A 0.000,B 0.000,C 90.000,E1 42.000} C_DIS
LIN {X -0.028,Y -474.296,Z 509.026,A 0.000,B 0.000,C 90.000,E1 40.744} C_DIS
LIN {X -0.007,Y -473.946,Z 509.021,A 0.000,B 0.000,C 90.000,E1 39.806} C_DIS
LIN {X -0.111,Y -473.287,Z 509.013,A 0.000,B 0.000,C 90.000,E1 38.257} C_DIS
LIN {X 0.143,Y -472.448,Z 509.004,A 0.000,B 0.000,C 90.000,E1 36.664} C_DIS
LIN {X 0.096,Y -471.569,Z 508.995,A 0.000,B 0.000,C 90.000,E1 35.105} C_DIS
LIN {X -0.074,Y -470.291,Z 508.985,A 0.000,B 0.000,C 90.000,E1 33.245} C_DIS
LIN {X 0.119,Y -468.855,Z 508.974,A 0.000,B 0.000,C 90.000,E1 31.337} C_DIS
LIN {X 0.024,Y -467.302,Z 508.964,A 0.000,B 0.000,C 90.000,E1 29.461} C_DIS
LIN {X -0.158,Y -465.718,Z 508.953,A 0.000,B 0.000,C 90.000,E1 27.590} C_DIS
LIN {X -0.015,Y -464.757,Z 508.946,A 0.000,B 0.000,C 90.000,E1 26.309} C_DIS
LIN {X 0.091,Y -463.151,Z 508.934,A 0.000,B 0.000,C 90.000,E1 24.079} C_DIS
LIN {X 0.047,Y -461.476,Z 508.918,A 0.000,B 0.000,C 90.000,E1 21.227} C_DIS
LIN {X -0.222,Y -460.464,Z 508.906,A 0.000,B 0.000,C 90.000,E1 19.033} C_DIS
LIN {X 0.025,Y -459.371,Z 508.890,A 0.000,B 0.000,C 90.000,E1 16.134} C_DIS
LIN {X 0.044,Y -458.953,Z 508.881,A 0.000,B 0.000,C 90.000,E1 14.537} C_DIS
LIN {X 0.081,Y -458.756,Z 508.865,A 0.000,B 0.000,C 90.000,E1 11.658} C_DIS
LIN {X -0.064,Y -459.041,Z 508.849,A 0.000,B 0.000,C 90.000,E1 8.803} C_DIS
LIN {X 0.105,Y -459.841,Z 508.833,A 0.000,B 0.000,C 90.000,E1 5.910} C_DIS
LIN {X 0.187,Y -460.946,Z 508.821,A 0.000,B 0.000,C 90.000,E1 3.669} C_DIS
LIN {X -0.187,Y -462.430,Z 508.808,A 0.000,B 0.000,C 90.000,E1 1.489} C_DIS
LIN {X 0.118,Y -465.000,Z 508.792,A 0.000,B 0.000,C 90.000,E1 358.511} C_DIS
LIN {X -0.144,Y -467.383,Z 508.780,A 0.000,B 0.000,C 90.000,E1 356.331} C_DIS
LIN {X 0.125,Y -469.313,Z 508.771,A 0.000,B 0.000,C 90.000,E1 354.723} C_DIS
LIN {X 0.194,Y -470.970,Z 508.764,A 0.000,B 0.000,C 90.000,E1 353.457} C_DIS
LIN {X 0.167,Y -472.996,Z 508.755,A 0.000,B 0.000,C 90.000,E1 351.894} C_DIS
LIN {X 0.005,Y -476.966,Z 508.740,A 0.000,B 0.000,C 90.000,E1 349.106} C_DIS
LIN {X -0.022,Y -480.429,Z 508.727,A 0.000,B 0.000,C 90.000,E1 346.937} C_DIS
LIN {X 0.146,Y -485.020,Z 508.714,A 0.000,B 0.000,C 90.000,E1 344.448} C_DIS
LIN {X 0.232,Y -488.724,Z 508.704,A 0.000,B 0.000,C 90.000,E1 342.598} C_DIS
LIN {X 0.079,Y -492.620,Z 508.693,A 0.000,B 0.000,C 90.000,E1 340.786} C_DIS
LIN {X 0.178,Y -496.456,Z 508.683,A 0.000,B 0.000,C 90.000,E1 338.954} C_DIS
LIN {X -0.239,Y -499.024,Z 508.677,A 0.000,B 0.000,C 90.000,E1 337.794} C_DIS
LIN {X 0.022,Y -501.495,Z 508.670,A 0.000,B 0.000,C 90.000,E1 336.561} C_DIS
LIN {X 0.063,Y -503.951,Z 508.663,A 0.000,B 0.000,C 90.000,E1 335.357} C_DIS
LIN {X -0.140,Y -507.412,Z 508.653,A 0.000,B 0.000,C 90.000,E1 333.589} C_DIS
LIN {X 0.190,Y -510.999,Z 508.643,A 0.000,B 0.000,C 90.000,E1 331.769} C_DIS
LIN {X -0.193,Y -513.970,Z 508.635,A 0.000,B 0.000,C 90.000,E1 330.333} C_DIS
LIN {X -0.270,Y -517.078,Z 508.627,A 0.000,B 0.000,C 90.000,E1 328.869} C_DIS
LIN {X 0.020,Y -521.365,Z 508.616,A 0.000,B 0.000,C 90.000,E1 326.786} C_DIS
LIN {X -0.171,Y -525.764,Z 508.604,A 0.000,B 0.000,C 90.000,E1 324.769} C_DIS
LIN {X 0.077,Y -529.529,Z 508.595,A 0.000,B 0.000,C 90.000,E1 323.004} C_DIS
LIN {X -0.116,Y -533.882,Z 508.583,A 0.000,B 0.000,C 90.000,E1 321.009} C_DIS
LIN {X 0.208,Y -536.929,Z 508.575,A 0.000,B 0.000,C 90.000,E1 319.542} C_DIS
LIN {X -0.233,Y -540.031,Z 508.567,A 0.000,B 0.000,C 90.000,E1 318.162} C_DIS
LIN {X -0.243,Y -543.703,Z 508.558,A 0.000,B 0.000,C 90.000,E1 316.458} C_DIS
LIN {X -0.192,Y -547.242,Z 508.549,A 0.000,B 0.000,C 90.000,E1 314.757} C_DIS
LIN {X -0.080,Y -550.154,Z 508.541,A 0.000,B 0.000,C 90.000,E1 313.338} C_DIS
LIN {X -0.216,Y -554.153,Z 508.530,A 0.000,B 0.000,C 90.000,E1 311.391} C_DIS
LIN {X 0.068,Y -557.032,Z 508.522,A 0.000,B 0.000,C 90.000,E1 309.967} C_DIS
LIN {X -0.033,Y -560.027,Z 508.514,A 0.000,B 0.000,C 90.000,E1 308.588} C_DIS
LIN {X -0.246,Y -563.433,Z 508.505,A 0.000,B 0.000,C 90.000,E1 306.950} C_DIS
LIN {X 0.081,Y -566.806,Z 508.496,A 0.000,B 0.000,C 90.000,E1 305.264} C_DIS
LIN {X 0.008,Y -570.235,Z 508.487,A 0.000,B 0.000,C 90.000,E1 303.627} C_DIS
LIN {X -0.159,Y -573.668,Z 508.478,A 0.000,B 0.000,C 90.000,E1 302.005} C_DIS
LIN {X 0.105,Y -576.422,Z 508.470,A 0.000,B 0.000,C 90.000,E1 300.620} C_DIS
LIN {X -0.076,Y -579.063,Z 508.463,A 0.000,B 0.000,C 90.000,E1 299.283} C_DIS
LIN {X 0.148,Y -582.265,Z 508.454,A 0.000,B 0.000,C 90.000,E1 297.641} C_DIS
LIN {X 0.148,Y -583.890,Z 508.448,A 0.000,B 0.000,C 90.000,E1 296.565} C_DIS
LIN {X -0.102,Y -584.617,Z 508.445,A 0.000,B 0.000,C 90.000,E1 296.052} C_DIS
LIN {X 0.309,Y -585.451,Z 508.440,A 0.000,B 0.000,C 90.000,E1 295.207} C_DIS
LIN {X -0.303,Y -585.965,Z 508.436,A 0.000,B 0.000,C 90.000,E1 294.463} C_DIS
LIN {X -0.009,Y -586.138,Z 508.433,A 0.000,B 0.000,C 90.000,E1 293.898} C_DIS
LIN {X -0.142,Y -586.780,Z 508.421,A 0.000,B 0.000,C 90.000,E1 291.770} C_DIS
LIN {X -0.108,Y -587.581,Z 508.413,A 0.000,B 0.000,C 90.000,E1 290.429} C_DIS
LIN {X 0.271,Y -588.053,Z 508.408,A 0.000,B 0.000,C 90.000,E1 289.322} C_DIS
LIN {X -0.100,Y -588.333,Z 508.402,A 0.000,B 0.000,C 90.000,E1 288.290} C_DIS
LIN {X 0.329,Y -588.489,Z 508.394,A 0.000,B 0.000,C 90.000,E1 286.913} C_DIS
LIN {X -0.215,Y -588.531,Z 508.388,A 0.000,B 0.000,C 90.000,E1 285.898} C_DIS
LIN {X -0.256,Y -588.492,Z 508.379,A 0.000,B 0.000,C 90.000,E1 284.300} C_DIS
LIN {X 0.017,Y -588.382,Z 508.372,A 0.000,B 0.000,C 90.000,E1 282.939} C_DIS
LIN {X -0.286,Y -588.232,Z 508.363,A 0.000,B 0.000,C 90.000,E1 281.366} C_DIS
LIN {X -0.323,Y -587.908,Z 508.353,A 0.000,B 0.000,C 90.000,E1 279.500} C_DIS
LIN {X 0.273,Y -587.590,Z 508.345,A 0.000,B 0.000,C 90.000,E1 278.106} C_DIS
LIN {X -0.145,Y -587.067,Z 508.336,A 0.000,B 0.000,C 90.000,E1 276.543} C_DIS
LIN {X 0.046,Y -586.596,Z 508.330,A 0.000,B 0.000,C 90.000,E1 275.454} C_DIS
LIN {X -0.107,Y -585.820,Z 508.323,A 0.000,B 0.000,C 90.000,E1 274.131} C_DIS
LIN {X -0.284,Y -584.808,Z 508.315,A 0.000,B 0.000,C 90.000,E1 272.808} C_DIS
LIN {X -0.114,Y -583.805,Z 508.310,A 0.000,B 0.000,C 90.000,E1 271.718} C_DIS
LIN {X 0.203,Y -582.441,Z 508.302,A 0.000,B 0.000,C 90.000,E1 270.344} C_DIS
LIN {X 0.090,Y -580.621,Z 508.293,A 0.000,B 0.000,C 90.000,E1 268.740} C_DIS
LIN {X 0.137,Y -578.294,Z 508.283,A 0.000,B 0.000,C 90.000,E1 266.846} C_DIS
LIN {X -0.205,Y -576.592,Z 508.275,A 0.000,B 0.000,C 90.000,E1 265.527} C_DIS
LIN {X -0.103,Y -575.167,Z 508.269,A 0.000,B 0.000,C 90.000,E1 264.432} C_DIS
LIN {X -0.270,Y -572.792,Z 508.260,A 0.000,B 0.000,C 90.000,E1 262.818} C_DIS
LIN {X 0.147,Y -570.183,Z 508.251,A 0.000,B 0.000,C 90.000,E1 261.141} C_DIS
LIN {X 0.035,Y -567.565,Z 508.242,A 0.000,B 0.000,C 90.000,E1 259.511} C_DIS
LIN {X -0.308,Y -565.258,Z 508.234,A 0.000,B 0.000,C 90.000,E1 258.173} C_DIS
LIN {X 0.096,Y -562.872,Z 508.227,A 0.000,B 0.000,C 90.000,E1 256.756} C_DIS
LIN {X 0.174,Y -560.865,Z 508.220,A 0.000,B 0.000,C 90.000,E1 255.644} C_DIS
LIN {X -0.186,Y -558.707,Z 508.214,A 0.000,B 0.000,C 90.000,E1 254.574} C_DIS
LIN {X 0.244,Y -555.817,Z 508.207,A 0.000,B 0.000,C 90.000,E1 253.142} C_DIS
LIN {X -0.163,Y -552.031,Z 508.197,A 0.000,B 0.000,C 90.000,E1 251.511} C_DIS
LIN {X 0.043,Y -549.384,Z 508.191,A 0.000,B 0.000,C 90.000,E1 250.369} C_DIS
LIN {X -0.320,Y -545.056,Z 508.182,A 0.000,B 0.000,C 90.000,E1 248.720} C_DIS
LIN {X -0.102,Y -541.313,Z 508.174,A 0.000,B 0.000,C 90.000,E1 247.283} C_DIS
LIN {X 0.055,Y -537.334,Z 508.166,A 0.000,B 0.000,C 90.000,E1 245.845} C_DIS
LIN {X -0.070,Y -534.027,Z 508.160,A 0.000,B 0.000,C 90.000,E1 244.717} C_DIS
LIN {X -0.015,Y -530.636,Z 508.153,A 0.000,B 0.000,C 90.000,E1 243.563} C_DIS
LIN {X -0.152,Y -525.353,Z 508.144,A 0.000,B 0.000,C 90.000,E1 241.847} C_DIS
LIN {X 0.078,Y -520.046,Z 508.134,A 0.000,B 0.000,C 90.000,E1 240.078} C_DIS
LIN {X -0.017,Y -516.468,Z 508.127,A 0.000,B 0.000,C 90.000,E1 238.918} C_DIS
LIN {X -0.073,Y -511.840,Z 508.119,A 0.000,B 0.000,C 90.000,E1 237.454} C_DIS
LIN {X -0.277,Y -508.051,Z 508.113,A 0.000,B 0.000,C 90.000,E1 236.294} C_DIS
LIN {X -0.168,Y -501.355,Z 508.101,A 0.000,B 0.000,C 90.000,E1 234.196} C_DIS
LIN {X -0.212,Y -491.468,Z 508.083,A 0.000,B 0.000,C 90.000,E1 230.884} C_DIS
LIN {X 0.249,Y -483.864,Z 508.067,A 0.000,B 0.000,C 90.000,E1 228.081} C_DIS
LIN {X -0.090,Y -479.849,Z 508.059,A 0.000,B 0.000,C 90.000,E1 226.581} C_DIS
LIN {X -0.279,Y -474.228,Z 508.047,A 0.000,B 0.000,C 90.000,E1 224.433} C_DIS
LIN {X -0.037,Y -469.595,Z 508.036,A 0.000,B 0.000,C 90.000,E1 222.528} C_DIS
LIN {X 0.125,Y -465.106,Z 508.026,A 0.000,B 0.000,C 90.000,E1 220.620} C_DIS
LIN {X -0.118,Y -460.888,Z 508.015,A 0.000,B 0.000,C 90.000,E1 218.749} C_DIS
LIN {X -0.011,Y -456.079,Z 508.003,A 0.000,B 0.000,C 90.000,E1 216.503} C_DIS
LIN {X 0.054,Y -451.461,Z 507.990,A 0.000,B 0.000,C 90.000,E1 214.246} C_DIS
LIN {X -0.132,Y -447.102,Z 507.978,A 0.000,B 0.000,C 90.000,E1 212.005} C_DIS
LIN {X -0.115,Y -443.497,Z 507.967,A 0.000,B 0.000,C 90.000,E1 210.050} C_DIS
LIN {X -0.199,Y -439.378,Z 507.954,A 0.000,B 0.000,C 90.000,E1 207.769} C_DIS
LIN {X 0.119,Y -437.053,Z 507.947,A 0.000,B 0.000,C 90.000,E1 206.411} C_DIS
LIN {X -0.149,Y -433.611,Z 507.936,A 0.000,B 0.000,C 90.000,E1 204.463} C_DIS
LIN {X -0.090,Y -430.271,Z 507.925,A 0.000,B 0.000,C 90.000,E1 202.461} C_DIS
LIN {X 0.120,Y -426.102,Z 507.910,A 0.000,B 0.000,C 90.000,E1 199.758} C_DIS
LIN {X -0.093,Y -422.344,Z 507.895,A 0.000,B 0.000,C 90.000,E1 197.094} C_DIS
LIN {X 0.131,Y -418.916,Z 507.880,A 0.000,B 0.000,C 90.000,E1 194.356} C_DIS
LIN {X -0.106,Y -416.119,Z 507.867,A 0.000,B 0.000,C 90.000,E1 192.007} C_DIS
LIN {X -0.138,Y -413.880,Z 507.855,A 0.000,B 0.000,C 90.000,E1 189.962} C_DIS
LIN {X 0.084,Y -411.401,Z 507.842,A 0.000,B 0.000,C 90.000,E1 187.530} C_DIS
LIN {X 0.180,Y -409.637,Z 507.832,A 0.000,B 0.000,C 90.000,E1 185.796} C_DIS
LIN {X 0.129,Y -406.679,Z 507.815,A 0.000,B 0.000,C 90.000,E1 182.694} C_DIS
LIN {X -0.019,Y -404.977,Z 507.802,A 0.000,B 0.000,C 90.000,E1 180.286} C_DIS
LIN {X -0.190,Y -403.761,Z 507.790,A 0.000,B 0.000,C 90.000,E1 178.224} C_DIS
LIN {X -0.074,Y -402.516,Z 507.771,A 0.000,B 0.000,C 90.000,E1 174.723} C_DIS
LIN {X 0.178,Y -402.171,Z 507.755,A 0.000,B 0.000,C 90.000,E1 171.894} C_DIS
LIN {X 0.154,Y -402.276,Z 507.744,A 0.000,B 0.000,C 90.000,E1 169.803} C_DIS
LIN {X -0.194,Y -402.696,Z 507.730,A 0.000,B 0.000,C 90.000,E1 167.409} C_DIS
LIN {X 0.123,Y -403.524,Z 507.714,A 0.000,B 0.000,C 90.000,E1 164.574} C_DIS
LIN {X -0.089,Y -404.813,Z 507.699,A 0.000,B 0.000,C 90.000,E1 161.819} C_DIS
LIN {X 0.160,Y -406.091,Z 507.687,A 0.000,B 0.000,C 90.000,E1 159.699} C_DIS
LIN {X -0.077,Y -408.294,Z 507.670,A 0.000,B 0.000,C 90.000,E1 156.613} C_DIS
LIN {X -0.047,Y -410.064,Z 507.659,A 0.000,B 0.000,C 90.000,E1 154.537} C_DIS
LIN {X 0.097,Y -411.505,Z 507.649,A 0.000,B 0.000,C 90.000,E1 152.794} C_DIS
LIN {X -0.088,Y -412.928,Z 507.639,A 0.000,B 0.000,C 90.000,E1 151.101} C_DIS
LIN {X -0.254,Y -414.265,Z 507.630,A 0.000,B 0.000,C 90.000,E1 149.410} C_DIS
LIN {X 0.022,Y -415.540,Z 507.620,A 0.000,B 0.000,C 90.000,E1 147.661} C_DIS
LIN {X -0.031,Y -416.686,Z 507.611,A 0.000,B 0.000,C 90.000,E1 145.960} C_DIS
LIN {X -0.044,Y -418.170,Z 507.598,A 0.000,B 0.000,C 90.000,E1 143.577} C_DIS
LIN {X -0.050,Y -418.814,Z 507.592,A 0.000,B 0.000,C 90.000,E1 142.557} C_DIS
LIN {X 0.154,Y -419.568,Z 507.584,A 0.000,B 0.000,C 90.000,E1 141.170} C_DIS
LIN {X 0.046,Y -420.284,Z 507.577,A 0.000,B 0.000,C 90.000,E1 139.828} C_DIS
LIN {X 0.035,Y -421.154,Z 507.566,A 0.000,B 0.000,C 90.000,E1 137.796} C_DIS
LIN {X -0.090,Y -421.537,Z 507.558,A 0.000,B 0.000,C 90.000,E1 136.458} C_DIS
LIN {X -0.016,Y -421.775,Z 507.549,A 0.000,B 0.000,C 90.000,E1 134.757} C_DIS
LIN {X -0.224,Y -421.830,Z 507.545,A 0.000,B 0.000,C 90.000,E1 134.109} C_DIS
LIN {X 0.261,Y -421.611,Z 507.537,A 0.000,B 0.000,C 90.000,E1 132.690} C_DIS
LIN {X 0.251,Y -421.259,Z 507.532,A 0.000,B 0.000,C 90.000,E1 131.676} C_DIS
LIN {X -0.156,Y -420.396,Z 507.524,A 0.000,B 0.000,C 90.000,E1 130.378} C_DIS
LIN {X -0.136,Y -419.598,Z 507.519,A 0.000,B 0.000,C 90.000,E1 129.358} C_DIS
LIN {X -0.053,Y -418.193,Z 507.509,A 0.000,B 0.000,C 90.000,E1 127.649} C_DIS
LIN {X 0.049,Y -416.434,Z 507.498,A 0.000,B 0.000,C 90.000,E1 125.678} C_DIS
LIN {X 0.166,Y -416.370,Z 507.498,A 0.000,B 0.000,C 90.000,E1 125.598} C_DIS
LIN {X 0.128,Y -416.367,Z 507.498,A 0.000,B 0.000,C 90.000,E1 125.598} C_DIS
LIN {X -0.080,Y -426.007,Z 507.477,A 0.000,B 0.000,C 90.000,E1 121.878} C_DIS
LIN {X -0.127,Y -430.998,Z 507.468,A 0.000,B 0.000,C 90.000,E1 120.207} C_DIS
LIN {X 0.017,Y -440.068,Z 507.448,A 0.000,B 0.000,C 90.000,E1 116.539} C_DIS
LIN {X 0.016,Y -444.852,Z 507.438,A 0.000,B 0.000,C 90.000,E1 114.899} C_DIS
LIN {X 0.275,Y -453.959,Z 507.417,A 0.000,B 0.000,C 90.000,E1 110.972} C_DIS
LIN {X 0.134,Y -457.432,Z 507.410,A 0.000,B 0.000,C 90.000,E1 109.704} C_DIS
LIN {X 0.225,Y -459.451,Z 507.404,A 0.000,B 0.000,C 90.000,E1 108.598} C_DIS
LIN {X 0.185,Y -459.617,Z 507.404,A 0.000,B 0.000,C 90.000,E1 108.598} C_DIS
LIN {X 0.086,Y -483.862,Z 507.400,A 0.000,B 0.000,C 90.000,E1 107.946} C_DIS
LIN {X 0.152,Y -494.293,Z 507.398,A 0.000,B 0.000,C 90.000,E1 107.638} C_DIS
LIN {X 0.018,Y -508.313,Z 507.396,A 0.000,B 0.000,C 90.000,E1 107.221} C_DIS
LIN {X 0.232,Y -522.381,Z 507.393,A 0.000,B 0.000,C 90.000,E1 106.732} C_DIS
LIN {X 0.011,Y -535.916,Z 507.390,A 0.000,B 0.000,C 90.000,E1 106.260} C_DIS
LIN {X -0.239,Y -542.308,Z 507.389,A 0.000,B 0.000,C 90.000,E1 106.024} C_DIS
LIN {X 0.074,Y -545.779,Z 507.388,A 0.000,B 0.000,C 90.000,E1 105.843} C_DIS
LIN {X -0.012,Y -552.312,Z 507.386,A 0.000,B 0.000,C 90.000,E1 105.552} C_DIS
LIN {X 0.227,Y -555.385,Z 507.386,A 0.000,B 0.000,C 90.000,E1 105.371} C_DIS
LIN {X 0.222,Y -558.077,Z 507.385,A 0.000,B 0.000,C 90.000,E1 105.245} C_DIS
LIN {X -0.193,Y -564.136,Z 507.383,A 0.000,B 0.000,C 90.000,E1 104.954} C_DIS
LIN {X 0.239,Y -570.004,Z 507.381,A 0.000,B 0.000,C 90.000,E1 104.537} C_DIS
LIN {X 0.163,Y -574.532,Z 507.379,A 0.000,B 0.000,C 90.000,E1 104.245} C_DIS
LIN {X 0.121,Y -580.376,Z 507.377,A 0.000,B 0.000,C 90.000,E1 103.828} C_DIS
LIN {X -0.198,Y -586.001,Z 507.374,A 0.000,B 0.000,C 90.000,E1 103.411} C_DIS
LIN {X -0.290,Y -592.721,Z 507.371,A 0.000,B 0.000,C 90.000,E1 102.827} C_DIS
LIN {X 0.114,Y -597.920,Z 507.368,A 0.000,B 0.000,C 90.000,E1 102.299} C_DIS
LIN {X 0.088,Y -605.090,Z 507.364,A 0.000,B 0.000,C 90.000,E1 101.535} C_DIS
LIN {X 0.188,Y -609.694,Z 507.361,A 0.000,B 0.000,C 90.000,E1 101.007} C_DIS
LIN {X 0.160,Y -614.153,Z 507.358,A 0.000,B 0.000,C 90.000,E1 100.489} C_DIS
LIN {X 0.103,Y -619.291,Z 507.355,A 0.000,B 0.000,C 90.000,E1 99.849} C_DIS
LIN {X 0.251,Y -623.233,Z 507.352,A 0.000,B 0.000,C 90.000,E1 99.321} C_DIS
LIN {X -0.151,Y -629.033,Z 507.347,A 0.000,B 0.000,C 90.000,E1 98.511} C_DIS
LIN {X -0.091,Y -633.120,Z 507.344,A 0.000,B 0.000,C 90.000,E1 97.871} C_DIS
LIN {X 0.307,Y -638.855,Z 507.338,A 0.000,B 0.000,C 90.000,E1 96.834} C_DIS
LIN {X -0.270,Y -642.163,Z 507.335,A 0.000,B 0.000,C 90.000,E1 96.258} C_DIS
LIN {X -0.061,Y -644.612,Z 507.332,A 0.000,B 0.000,C 90.000,E1 95.739} C_DIS
LIN {X -0.247,Y -649.283,Z 507.326,A 0.000,B 0.000,C 90.000,E1 94.759} C_DIS
LIN {X -0.215,Y -652.461,Z 507.322,A 0.000,B 0.000,C 90.000,E1 94.012} C_DIS
LIN {X 0.014,Y -654.409,Z 507.319,A 0.000,B 0.000,C 90.000,E1 93.498} C_DIS
LIN {X 0.099,Y -656.857,Z 507.315,A 0.000,B 0.000,C 90.000,E1 92.751} C_DIS
LIN {X -0.289,Y -658.289,Z 507.313,A 0.000,B 0.000,C 90.000,E1 92.293} C_DIS
LIN {X 0.014,Y -659.486,Z 507.310,A 0.000,B 0.000,C 90.000,E1 91.776} C_DIS
LIN {X 0.303,Y -660.490,Z 507.307,A 0.000,B 0.000,C 90.000,E1 91.260} C_DIS
LIN {X -0.238,Y -661.402,Z 507.303,A 0.000,B 0.000,C 90.000,E1 90.573} C_DIS
LIN {X 0.069,Y -661.787,Z 507.300,A 0.000,B 0.000,C 90.000,E1 90.057} C_DIS
LIN {X 0.205,Y -661.765,Z 507.296,A 0.000,B 0.000,C 90.000,E1 89.312} C_DIS
LIN {X -0.148,Y -661.582,Z 507.294,A 0.000,B 0.000,C 90.000,E1 88.854} C_DIS
LIN {X 0.159,Y -661.175,Z 507.291,A 0.000,B 0.000,C 90.000,E1 88.339} C_DIS
LIN {X -0.176,Y -660.575,Z 507.288,A 0.000,B 0.000,C 90.000,E1 87.879} C_DIS
LIN {X -0.247,Y -658.705,Z 507.283,A 0.000,B 0.000,C 90.000,E1 86.906} C_DIS
LIN {X 0.071,Y -657.580,Z 507.280,A 0.000,B 0.000,C 90.000,E1 86.388} C_DIS
LIN {X -0.268,Y -656.224,Z 507.277,A 0.000,B 0.000,C 90.000,E1 85.927} C_DIS
LIN {X 0.287,Y -652.894,Z 507.272,A 0.000,B 0.000,C 90.000,E1 84.894} C_DIS
LIN {X -0.075,Y -650.985,Z 507.269,A 0.000,B 0.000,C 90.000,E1 84.432} C_DIS
LIN {X -0.024,Y -647.751,Z 507.265,A 0.000,B 0.000,C 90.000,E1 83.685} C_DIS
LIN {X 0.227,Y -645.369,Z 507.262,A 0.000,B 0.000,C 90.000,E1 83.166} C_DIS
LIN {X -0.010,Y -641.733,Z 507.258,A 0.000,B 0.000,C 90.000,E1 82.470} C_DIS
LIN {X -0.114,Y -636.841,Z 507.253,A 0.000,B 0.000,C 90.000,E1 81.602} C_DIS
LIN {X -0.278,Y -631.329,Z 507.248,A 0.000,B 0.000,C 90.000,E1 80.735} C_DIS
LIN {X -0.156,Y -626.252,Z 507.244,A 0.000,B 0.000,C 90.000,E1 79.982} C_DIS
LIN {X 0.039,Y -620.859,Z 507.240,A 0.000,B 0.000,C 90.000,E1 79.218} C_DIS
LIN {X -0.148,Y -614.736,Z 507.236,A 0.000,B 0.000,C 90.000,E1 78.465} C_DIS
LIN {X -0.087,Y -609.176,Z 507.232,A 0.000,B 0.000,C 90.000,E1 77.813} C_DIS
LIN {X 0.019,Y -604.358,Z 507.229,A 0.000,B 0.000,C 90.000,E1 77.285} C_DIS
LIN {X 0.143,Y -599.235,Z 507.227,A 0.000,B 0.000,C 90.000,E1 76.769} C_DIS
LIN {X 0.060,Y -592.400,Z 507.223,A 0.000,B 0.000,C 90.000,E1 76.172} C_DIS
LIN {X -0.002,Y -588.273,Z 507.221,A 0.000,B 0.000,C 90.000,E1 75.825} C_DIS
LIN {X -0.340,Y -582.334,Z 507.219,A 0.000,B 0.000,C 90.000,E1 75.408} C_DIS
LIN {X 0.120,Y -576.200,Z 507.216,A 0.000,B 0.000,C 90.000,E1 74.936} C_DIS
LIN {X 0.271,Y -571.265,Z 507.215,A 0.000,B 0.000,C 90.000,E1 74.629} C_DIS
LIN {X -0.206,Y -564.926,Z 507.213,A 0.000,B 0.000,C 90.000,E1 74.338} C_DIS
LIN {X 0.169,Y -559.741,Z 507.212,A 0.000,B 0.000,C 90.000,E1 74.047} C_DIS
LIN {X -0.192,Y -554.439,Z 507.210,A 0.000,B 0.000,C 90.000,E1 73.850} C_DIS
LIN {X 0.027,Y -546.860,Z 507.209,A 0.000,B 0.000,C 90.000,E1 73.559} C_DIS
LIN {X 0.057,Y -541.458,Z 507.208,A 0.000,B 0.000,C 90.000,E1 73.378} C_DIS
LIN {X -0.073,Y -533.509,Z 507.207,A 0.000,B 0.000,C 90.000,E1 73.196} C_DIS
LIN {X -0.210,Y -527.597,Z 507.206,A 0.000,B 0.000,C 90.000,E1 73.087} C_DIS
LIN {X 0.229,Y -519.477,Z 507.205,A 0.000,B 0.000,C 90.000,E1 72.906} C_DIS
LIN {X -0.124,Y -503.508,Z 507.204,A 0.000,B 0.000,C 90.000,E1 72.725} C_DIS
LIN {X 0.101,Y -494.024,Z 507.203,A 0.000,B 0.000,C 90.000,E1 72.598} C_DIS
LIN {X -0.170,Y -475.174,Z 507.203,A 0.000,B 0.000,C 90.000,E1 72.489} C_DIS
LIN {X -0.212,Y -474.541,Z 507.203,A 0.000,B 0.000,C 90.000,E1 72.489} C_DIS
LIN {X 0.134,Y -474.075,Z 507.200,A 0.000,B 0.000,C 90.000,E1 72.000} C_DIS
LIN {X 0.164,Y -465.514,Z 507.172,A 0.000,B 0.000,C 90.000,E1 66.975} C_DIS
LIN {X -0.058,Y -457.066,Z 507.149,A 0.000,B 0.000,C 90.000,E1 62.871} C_DIS
LIN {X 0.051,Y -455.483,Z 507.144,A 0.000,B 0.000,C 90.000,E1 61.897} C_DIS
LIN {X 0.073,Y -448.476,Z 507.127,A 0.000,B 0.000,C 90.000,E1 58.869} C_DIS
LIN {X 0.033,Y -448.484,Z 507.127,A 0.000,B 0.000,C 90.000,E1 58.869} C_DIS
LIN {X 0.126,Y -453.761,Z 507.120,A 0.000,B 0.000,C 90.000,E1 57.533} C_DIS
LIN {X -0.083,Y -456.698,Z 507.115,A 0.000,B 0.000,C 90.000,E1 56.755} C_DIS
LIN {X -0.141,Y -459.882,Z 507.110,A 0.000,B 0.000,C 90.000,E1 55.801} C_DIS
LIN {X 0.096,Y -462.643,Z 507.105,A 0.000,B 0.000,C 90.000,E1 54.815} C_DIS
LIN {X -0.032,Y -464.280,Z 507.101,A 0.000,B 0.000,C 90.000,E1 54.196} C_DIS
LIN {X -0.116,Y -466.414,Z 507.096,A 0.000,B 0.000,C 90.000,E1 53.256} C_DIS
LIN {X 0.198,Y -468.194,Z 507.091,A 0.000,B 0.000,C 90.000,E1 52.271} C_DIS
LIN {X 0.020,Y -469.257,Z 507.087,A 0.000,B 0.000,C 90.000,E1 51.662} C_DIS
LIN {X 0.203,Y -471.367,Z 507.078,A 0.000,B 0.000,C 90.000,E1 50.070} C_DIS
LIN {X -0.087,Y -472.704,Z 507.071,A 0.000,B 0.000,C 90.000,E1 48.852} C_DIS
LIN {X -0.133,Y -473.516,Z 507.066,A 0.000,B 0.000,C 90.000,E1 47.919} C_DIS
LIN {X -0.166,Y -474.191,Z 507.061,A 0.000,B 0.000,C 90.000,E1 46.986} C_DIS
LIN {X -0.195,Y -474.738,Z 507.056,A 0.000,B 0.000,C 90.000,E1 46.053} C_DIS
LIN {X 0.112,Y -475.164,Z 507.051,A 0.000,B 0.000,C 90.000,E1 45.081} C_DIS
LIN {X -0.144,Y -475.513,Z 507.044,A 0.000,B 0.000,C 90.000,E1 43.866} C_DIS
LIN {X -0.053,Y -475.572,Z 507.037,A 0.000,B 0.000,C 90.000,E1 42.609} C_DIS
LIN {X 0.033,Y -475.330,Z 507.030,A 0.000,B 0.000,C 90.000,E1 41.353} C_DIS
LIN {X 0.063,Y -475.048,Z 507.025,A 0.000,B 0.000,C 90.000,E1 40.415} C_DIS
LIN {X 0.069,Y -474.247,Z 507.014,A 0.000,B 0.000,C 90.000,E1 38.543} C_DIS
LIN {X -0.037,Y -473.425,Z 507.006,A 0.000,B 0.000,C 90.000,E1 36.996} C_DIS
LIN {X -0.073,Y -472.524,Z 506.997,A 0.000,B 0.000,C 90.000,E1 35.438} C_DIS
LIN {X -0.173,Y -471.662,Z 506.990,A 0.000,B 0.000,C 90.000,E1 34.199} C_DIS
LIN {X -0.283,Y -470.757,Z 506.983,A 0.000,B 0.000,C 90.000,E1 32.959} C_DIS
LIN {X 0.153,Y -469.571,Z 506.974,A 0.000,B 0.000,C 90.000,E1 31.337} C_DIS
LIN {X 0.073,Y -467.968,Z 506.964,A 0.000,B 0.000,C 90.000,E1 29.461} C_DIS
LIN {X -0.093,Y -466.350,Z 506.953,A 0.000,B 0.000,C 90.000,E1 27.590} C_DIS
LIN {X 0.195,Y -465.093,Z 506.944,A 0.000,B 0.000,C 90.000,E1 25.976} C_DIS
LIN {X 0.180,Y -463.687,Z 506.934,A 0.000,B 0.000,C 90.000,E1 24.079} C_DIS
LIN {X -0.130,Y -462.291,Z 506.922,A 0.000,B 0.000,C 90.000,E1 21.897} C_DIS
LIN {X -0.069,Y -461.508,Z 506.913,A 0.000,B 0.000,C 90.000,E1 20.301} C_DIS
LIN {X 0.172,Y -460.641,Z 506.902,A 0.000,B 0.000,C 90.000,E1 18.362} C_DIS
LIN {X 0.161,Y -459.825,Z 506.890,A 0.000,B 0.000,C 90.000,E1 16.134} C_DIS
LIN {X -0.031,Y -459.281,Z 506.879,A 0.000,B 0.000,C 90.000,E1 14.245} C_DIS
LIN {X -0.211,Y -459.092,Z 506.865,A 0.000,B 0.000,C 90.000,E1 11.715} C_DIS
LIN {X 0.104,Y -459.322,Z 506.849,A 0.000,B 0.000,C 90.000,E1 8.803} C_DIS
LIN {X -0.185,Y -459.834,Z 506.837,A 0.000,B 0.000,C 90.000,E1 6.606} C_DIS
LIN {X 0.174,Y -461.010,Z 506.822,A 0.000,B 0.000,C 90.000,E1 4.012} C_DIS
LIN {X 0.033,Y -462.158,Z 506.812,A 0.000,B 0.000,C 90.000,E1 2.121} C_DIS
LIN {X 0.000,Y -463.789,Z 506.800,A 0.000,B 0.000,C 90.000,E1 360.000} C_DIS
LIN {X 0.114,Y -465.823,Z 506.788,A 0.000,B 0.000,C 90.000,E1 357.879} C_DIS
LIN {X -0.137,Y -467.571,Z 506.780,A 0.000,B 0.000,C 90.000,E1 356.331} C_DIS
LIN {X 0.137,Y -469.473,Z 506.771,A 0.000,B 0.000,C 90.000,E1 354.723} C_DIS
LIN {X 0.023,Y -471.517,Z 506.762,A 0.000,B 0.000,C 90.000,E1 353.166} C_DIS
LIN {X 0.183,Y -473.151,Z 506.755,A 0.000,B 0.000,C 90.000,E1 351.894} C_DIS
LIN {X -0.131,Y -477.563,Z 506.738,A 0.000,B 0.000,C 90.000,E1 348.814} C_DIS
LIN {X -0.143,Y -481.129,Z 506.726,A 0.000,B 0.000,C 90.000,E1 346.645} C_DIS
LIN {X 0.176,Y -485.211,Z 506.714,A 0.000,B 0.000,C 90.000,E1 344.448} C_DIS
LIN {X -0.214,Y -488.320,Z 506.705,A 0.000,B 0.000,C 90.000,E1 342.960} C_DIS
LIN {X 0.119,Y -492.841,Z 506.693,A 0.000,B 0.000,C 90.000,E1 340.786} C_DIS
LIN {X 0.222,Y -496.697,Z 506.683,A 0.000,B 0.000,C 90.000,E1 338.954} C_DIS
LIN {X -0.191,Y -499.295,Z 506.677,A 0.000,B 0.000,C 90.000,E1 337.794} C_DIS
LIN {X 0.076,Y -501.795,Z 506.670,A 0.000,B 0.000,C 90.000,E1 336.561} C_DIS
LIN {X -0.258,Y -504.814,Z 506.662,A 0.000,B 0.000,C 90.000,E1 335.101} C_DIS
LIN {X 0.239,Y -508.329,Z 506.652,A 0.000,B 0.000,C 90.000,E1 333.256} C_DIS
LIN {X 0.262,Y -511.360,Z 506.643,A 0.000,B 0.000,C 90.000,E1 331.769} C_DIS
LIN {X 0.238,Y -514.938,Z 506.634,A 0.000,B 0.000,C 90.000,E1 329.999} C_DIS
LIN {X -0.182,Y -517.493,Z 506.627,A 0.000,B 0.000,C 90.000,E1 328.869} C_DIS
LIN {X 0.118,Y -521.830,Z 506.616,A 0.000,B 0.000,C 90.000,E1 326.786} C_DIS
LIN {X -0.060,Y -526.290,Z 506.604,A 0.000,B 0.000,C 90.000,E1 324.769} C_DIS
LIN {X -0.222,Y -530.087,Z 506.595,A 0.000,B 0.000,C 90.000,E1 323.050} C_DIS
LIN {X 0.028,Y -533.857,Z 506.585,A 0.000,B 0.000,C 90.000,E1 321.295} C_DIS
LIN {X 0.013,Y -536.348,Z 506.579,A 0.000,B 0.000,C 90.000,E1 320.150} C_DIS
LIN {X -0.070,Y -540.692,Z 506.568,A 0.000,B 0.000,C 90.000,E1 318.162} C_DIS
LIN {X -0.064,Y -544.406,Z 506.558,A 0.000,B 0.000,C 90.000,E1 316.458} C_DIS
LIN {X 0.004,Y -547.974,Z 506.549,A 0.000,B 0.000,C 90.000,E1 314.757} C_DIS
LIN {X 0.092,Y -550.288,Z 506.542,A 0.000,B 0.000,C 90.000,E1 313.623} C_DIS
LIN {X 0.189,Y -551.993,Z 506.538,A 0.000,B 0.000,C 90.000,E1 312.771} C_DIS
LIN {X 0.014,Y -554.921,Z 506.530,A 0.000,B 0.000,C 90.000,E1 311.391} C_DIS
LIN {X -0.113,Y -557.814,Z 506.522,A 0.000,B 0.000,C 90.000,E1 310.011} C_DIS
LIN {X -0.122,Y -560.790,Z 506.515,A 0.000,B 0.000,C 90.000,E1 308.624} C_DIS
LIN {X 0.141,Y -564.811,Z 506.504,A 0.000,B 0.000,C 90.000,E1 306.664} C_DIS
LIN {X 0.033,Y -568.220,Z 506.495,A 0.000,B 0.000,C 90.000,E1 305.025} C_DIS
LIN {X 0.139,Y -571.676,Z 506.486,A 0.000,B 0.000,C 90.000,E1 303.372} C_DIS
LIN {X 0.179,Y -574.553,Z 506.478,A 0.000,B 0.000,C 90.000,E1 302.005} C_DIS
LIN {X -0.036,Y -577.302,Z 506.470,A 0.000,B 0.000,C 90.000,E1 300.669} C_DIS
LIN {X -0.209,Y -579.927,Z 506.463,A 0.000,B 0.000,C 90.000,E1 299.333} C_DIS
LIN {X -0.114,Y -582.560,Z 506.455,A 0.000,B 0.000,C 90.000,E1 297.975} C_DIS
LIN {X 0.155,Y -584.260,Z 506.449,A 0.000,B 0.000,C 90.000,E1 296.873} C_DIS
LIN {X -0.218,Y -585.354,Z 506.445,A 0.000,B 0.000,C 90.000,E1 296.104} C_DIS
LIN {X -0.053,Y -586.266,Z 506.440,A 0.000,B 0.000,C 90.000,E1 295.283} C_DIS
LIN {X 0.124,Y -586.893,Z 506.436,A 0.000,B 0.000,C 90.000,E1 294.463} C_DIS
LIN {X 0.142,Y -587.656,Z 506.426,A 0.000,B 0.000,C 90.000,E1 292.589} C_DIS
LIN {X 0.287,Y -588.559,Z 506.417,A 0.000,B 0.000,C 90.000,E1 290.972} C_DIS
LIN {X -0.202,Y -589.207,Z 506.409,A 0.000,B 0.000,C 90.000,E1 289.685} C_DIS
LIN {X 0.001,Y -589.593,Z 506.403,A 0.000,B 0.000,C 90.000,E1 288.598} C_DIS
LIN {X -0.108,Y -589.816,Z 506.396,A 0.000,B 0.000,C 90.000,E1 287.275} C_DIS
LIN {X -0.216,Y -589.931,Z 506.389,A 0.000,B 0.000,C 90.000,E1 285.953} C_DIS
LIN {X 0.081,Y -589.943,Z 506.381,A 0.000,B 0.000,C 90.000,E1 284.592} C_DIS
LIN {X -0.069,Y -589.885,Z 506.372,A 0.000,B 0.000,C 90.000,E1 283.008} C_DIS
LIN {X 0.051,Y -589.740,Z 506.362,A 0.000,B 0.000,C 90.000,E1 281.130} C_DIS
LIN {X -0.217,Y -589.491,Z 506.353,A 0.000,B 0.000,C 90.000,E1 279.557} C_DIS
LIN {X -0.176,Y -589.200,Z 506.346,A 0.000,B 0.000,C 90.000,E1 278.219} C_DIS
LIN {X 0.201,Y -588.612,Z 506.335,A 0.000,B 0.000,C 90.000,E1 276.315} C_DIS
LIN {X 0.076,Y -587.941,Z 506.328,A 0.000,B 0.000,C 90.000,E1 274.992} C_DIS
LIN {X -0.250,Y -587.274,Z 506.322,A 0.000,B 0.000,C 90.000,E1 273.955} C_DIS
LIN {X 0.145,Y -586.194,Z 506.314,A 0.000,B 0.000,C 90.000,E1 272.579} C_DIS
LIN {X -0.064,Y -584.862,Z 506.307,A 0.000,B 0.000,C 90.000,E1 271.260} C_DIS
LIN {X 0.093,Y -583.695,Z 506.301,A 0.000,B 0.000,C 90.000,E1 270.172} C_DIS
LIN {X 0.005,Y -581.847,Z 506.292,A 0.000,B 0.000,C 90.000,E1 268.568} C_DIS
LIN {X 0.081,Y -579.429,Z 506.282,A 0.000,B 0.000,C 90.000,E1 266.674} C_DIS
LIN {X -0.246,Y -577.678,Z 506.274,A 0.000,B 0.000,C 90.000,E1 265.355} C_DIS
LIN {X -0.131,Y -576.173,Z 506.268,A 0.000,B 0.000,C 90.000,E1 264.261} C_DIS
LIN {X 0.161,Y -574.123,Z 506.261,A 0.000,B 0.000,C 90.000,E1 262.875} C_DIS
LIN {X 0.042,Y -571.462,Z 506.251,A 0.000,B 0.000,C 90.000,E1 261.254} C_DIS
LIN {X -0.141,Y -568.813,Z 506.242,A 0.000,B 0.000,C 90.000,E1 259.634} C_DIS
LIN {X 0.201,Y -566.425,Z 506.235,A 0.000,B 0.000,C 90.000,E1 258.229} C_DIS
LIN {X -0.218,Y -564.513,Z 506.229,A 0.000,B 0.000,C 90.000,E1 257.173} C_DIS
LIN {X 0.176,Y -561.973,Z 506.221,A 0.000,B 0.000,C 90.000,E1 255.755} C_DIS
LIN {X -0.163,Y -559.783,Z 506.215,A 0.000,B 0.000,C 90.000,E1 254.685} C_DIS
LIN {X 0.134,Y -556.869,Z 506.207,A 0.000,B 0.000,C 90.000,E1 253.268} C_DIS
LIN {X 0.163,Y -553.673,Z 506.199,A 0.000,B 0.000,C 90.000,E1 251.873} C_DIS
LIN {X -0.127,Y -551.071,Z 506.193,A 0.000,B 0.000,C 90.000,E1 250.786} C_DIS
LIN {X 0.056,Y -548.216,Z 506.187,A 0.000,B 0.000,C 90.000,E1 249.645} C_DIS
LIN {X -0.138,Y -543.805,Z 506.178,A 0.000,B 0.000,C 90.000,E1 247.975} C_DIS
LIN {X -0.173,Y -540.694,Z 506.171,A 0.000,B 0.000,C 90.000,E1 246.847} C_DIS
LIN {X 0.243,Y -537.451,Z 506.165,A 0.000,B 0.000,C 90.000,E1 245.665} C_DIS
LIN {X -0.167,Y -533.231,Z 506.157,A 0.000,B 0.000,C 90.000,E1 244.280} C_DIS
LIN {X 0.165,Y -530.657,Z 506.152,A 0.000,B 0.000,C 90.000,E1 243.384} C_DIS
LIN {X 0.267,Y -525.364,Z 506.143,A 0.000,B 0.000,C 90.000,E1 241.641} C_DIS
LIN {X 0.167,Y -519.106,Z 506.131,A 0.000,B 0.000,C 90.000,E1 239.616} C_DIS
LIN {X -0.287,Y -514.547,Z 506.123,A 0.000,B 0.000,C 90.000,E1 238.201} C_DIS
LIN {X -0.110,Y -509.862,Z 506.115,A 0.000,B 0.000,C 90.000,E1 236.707} C_DIS
LIN {X 0.045,Y -503.119,Z 506.103,A 0.000,B 0.000,C 90.000,E1 234.609} C_DIS
LIN {X -0.250,Y -497.448,Z 506.093,A 0.000,B 0.000,C 90.000,E1 232.844} C_DIS
LIN {X -0.214,Y -491.263,Z 506.082,A 0.000,B 0.000,C 90.000,E1 230.723} C_DIS
LIN {X 0.105,Y -484.498,Z 506.068,A 0.000,B 0.000,C 90.000,E1 228.243} C_DIS
LIN {X 0.127,Y -480.455,Z 506.060,A 0.000,B 0.000,C 90.000,E1 226.701} C_DIS
LIN {X 0.167,Y -475.586,Z 506.049,A 0.000,B 0.000,C 90.000,E1 224.838} C_DIS
LIN {X -0.137,Y -470.165,Z 506.037,A 0.000,B 0.000,C 90.000,E1 222.690} C_DIS
LIN {X -0.142,Y -464.191,Z 506.023,A 0.000,B 0.000,C 90.000,E1 220.172} C_DIS
LIN {X 0.210,Y -460.683,Z 506.014,A 0.000,B 0.000,C 90.000,E1 218.543} C_DIS
LIN {X 0.207,Y -457.280,Z 506.005,A 0.000,B 0.000,C 90.000,E1 216.950} C_DIS
LIN {X 0.032,Y -451.983,Z 505.991,A 0.000,B 0.000,C 90.000,E1 214.405} C_DIS
LIN {X 0.181,Y -447.029,Z 505.977,A 0.000,B 0.000,C 90.000,E1 211.799} C_DIS
LIN {X -0.091,Y -444.021,Z 505.968,A 0.000,B 0.000,C 90.000,E1 210.207} C_DIS
LIN {X 0.058,Y -439.870,Z 505.955,A 0.000,B 0.000,C 90.000,E1 207.897} C_DIS
LIN {X -0.205,Y -437.557,Z 505.948,A 0.000,B 0.000,C 90.000,E1 206.616} C_DIS
LIN {X 0.124,Y -434.091,Z 505.937,A 0.000,B 0.000,C 90.000,E1 204.591} C_DIS
LIN {X -0.204,Y -430.733,Z 505.926,A 0.000,B 0.000,C 90.000,E1 202.642} C_DIS
